// TIA Portal project "PLC_ScadaIT" (V15)

(* hardware
DEVICE "S71500/ET200MP station_1"  S7-1500 station
   slot 0: "Rail_0"  Rack  6ES7 590-1***0-0AA0
   slot 1: "PLC_CENTRAL.TAKT"  CPU 1516-3 PN/DP  6ES7 516-3AN01-0AB0  V2.5
      slot 3: "CPU display_1"  6ES7591-1BA00-0AA0
DEVICE "HMI_CENTRAL.TAKT"  TP900 Comfort
   slot 0: "HMI"  HMI  6AV2 124-0JC01-0AX0  13.0.1.0
   slot 1: "HMI_RT_1"  TP900 Comfort  6AV2 124-0JC01-0AX0  13.0.1.0
   slot 5: "HMI_CENTRAL.TAKT.IE_CP_1"  PROFINET Interface
      slot 1: "PROFINET Interface_1"  PROFINET Interface
         slot 1: "Port_1"  Port
         slot 2: "Port_2"  Port
   slot 7: "HMI_CENTRAL.TAKT.MPI/DP_CP_1"  MPI/DP Interface
*)

// ===== PLC "PLC_CENTRAL.TAKT"  CPU 1516-3 PN/DP =====

VAR_GLOBAL   // PLC tag table "Default tag table"
   "Clock_Byte" AT %MB0 : Byte;   // Byte de Clock
   "Clock_10Hz" AT %M0.0 : Bool;   // 0.1 Segundo
   "Clock_5Hz" AT %M0.1 : Bool;   // 0.2 Segundo
   "Clock_2.5Hz" AT %M0.2 : Bool;   // 0.4 Segundo
   "Clock_2Hz" AT %M0.3 : Bool;   // 0.5 Segundo
   "Clock_1.25Hz" AT %M0.4 : Bool;   // 0.8 Segundo
   "Clock_1Hz" AT %M0.5 : Bool;   // 1.0 Segundo
   "Clock_0.625Hz" AT %M0.6 : Bool;   // 1.6 Segundo
   "Clock_0.5Hz" AT %M0.7 : Bool;   // 2 Segundo
   "OFF" AT %M1.0 : Bool;   // First Scan
   "STATUS_PUT_DOCK" AT %MW603 : Word;
   "System_Byte" AT %MB1 : Byte;
   "DiagStatusUpdate" AT %M1.1 : Bool;
   "AlwaysTRUE" AT %M1.2 : Bool;
   "AlwaysFALSE" AT %M1.3 : Bool;
   "JOOJ" AT %M2.0 : Bool;
END_VAR

TYPE "Line_ReadInformation"
VERSION : 0.1
   STRUCT
      AndonExterno : Bool;   // Sinal recebido via sistema (celular)
      AndonP1 : Bool;   // Botão de andon do posto 1
      AndonP2 : Bool;   // Botão de andon do posto 2
      AndonP3 : Bool;   // Botão de andon do posto 3
      AndonP4 : Bool;   // Botão de andon do posto 4
      AndonP5 : Bool;   // Botão de andon do posto 5
      AndonP6 : Bool;   // Botão de andon do posto 6
      SensorFimDeLinha : Bool;   // Sensor RetroReflexivo do último posto
      EmergênciaP1 : Bool;   // Botão de emergência do posto 1
      EmergênciaP2 : Bool;   // Botão de emergência do posto 2
      EmergênciaP3 : Bool;   // Botão de emergência do posto 3
      EmergênciaP4 : Bool;   // Botão de emergência do posto 4
      EmergênciaP5 : Bool;   // Botão de emergência do posto 5
      EmergênciaP6 : Bool;   // Botão de emergência do posto 6
      StartRecebido : Bool;   // Confirma o recebimento do sinal de start
   END_STRUCT;
END_TYPE

TYPE "Agv.Database"
   STRUCT
      Emergencia : Bool;   // Botao de Emergecencia
      Warning : Bool;   // Area de Warning do Scanner
      Safety : Bool;   // Area de Safety do Scanner
      ConectarTakt : Bool;   // 0 - Desconectado / 1 - Conectado
      Rodando : Bool;
      Falha : Bool;
      AutomaticoManual : Byte;   // 1 - Manual / 2 - Automatico
      VelocidadeAtual : Int;   // Velocidade Atual
      Posto : Byte;   // Posto em que o AGV está
      Comando : Byte;   // Ultimo comando
      Velocidade : Byte;   // Velocidade Setada
      Processo : Byte;   // 1 - Ecu / 2 - SKD
      "Erros.Agv" : Byte;   // 0 á 256, cada numero um erro. 1 - Tudo Ok
      "Erros.Pgv" : Byte;   // 0 á 256, cada numero um erro. 1 - Tudo Ok
      "Erros.Rfid" : Byte;   // 0 á 256, cada numero um erro. 1 - Tudo Ok
      "Erros.MotorPasso" : Byte;   // 0 á 256, cada numero um erro. 1 - Tudo Ok
      "Erros.IOLink" : Byte;   // 0 á 256, cada numero um erro. 1 - Tudo Ok
      "Erros.Comunicacao" : Byte;   // 0 á 256, cada numero um erro. 1 - Tudo Ok
      Reservado : Byte;   // Reservado
      Reservado_1 : Byte;   // Reservado
      Reservado_2 : Byte;   // Reservado
      Reservado_3 : Byte;   // Reservado
      Reservado_4 : Byte;   // Reservado
      Reservado_5 : Byte;   // Reservado
      Reservado_6 : Byte;   // Reservado
      Reservado_7 : Byte;   // Reservado
      Reservado_8 : Byte;   // Reservado
   END_STRUCT;
END_TYPE

TYPE "Scada.Datebase"
   STRUCT
      Turnos : Struct
         Inicio : Array[0..2] of Time_Of_Day;
         Fim : Array[0..2] of Time_Of_Day;
      END_STRUCT;
      Paradas_Programadas : Struct
         Inicio : Array[0..5] of Time_Of_Day;
         Fim : Array[0..5] of Time_Of_Day;
      END_STRUCT;
      Dias_Da_Semana : Array[0..6] of Bool;
      ParametrosTakt : Array[0..2] of Struct
         Tempo_Takt : Int;
         ObjetivoTurno : Int;
      END_STRUCT;
      DiaDaSemana : Int;
   END_STRUCT;
   // // Dias_Da_Semana[0] : Segunda-Feira
   // // Dias_Da_Semana[1] : Terça-Feira
   // // Dias_Da_Semana[2] : Quarta-Feira
   // // Dias_Da_Semana[3] : Quinta-Feira
   // // Dias_Da_Semana[4] : Sexta-Feira
   // // Dias_Da_Semana[5] : Sabado
   // // Dias_Da_Semana[6] : Domingo
   // // ParametrosTakt[0] : Parametros do Takt do 1 turno
   // // ParametrosTakt[1] : Parametros do Takt do 2 turno
   // // ParametrosTakt[2] : Parametros do Takt do 3 turno
   // // Turnos.Inicio[0] : Incio 1 Turno
   // // Turnos.Inicio[1] : Incio 2 Turno
   // // Turnos.Inicio[2] : Incio 3 Turno
   // // Turnos.Fim[0] : Fim 1 Turno
   // // Turnos.Fim[1] : Fim 2 Turno
   // // Turnos.Fim[2] : Fim 3 Turno
   // // Paradas_Programadas.Inicio[0] : Inicio Parada Programada 1
   // // Paradas_Programadas.Inicio[1] : Inicio Parada Programada 2
   // // Paradas_Programadas.Fim[0] : Fim Parada Programada 1
   // // Paradas_Programadas.Inicio[2] : Inicio Parada Programada 3
   // // Paradas_Programadas.Inicio[3] : Inicio Parada Programada 4
   // // Paradas_Programadas.Inicio[4] : Inicio Parada Programada 5
   // // Paradas_Programadas.Inicio[5] : Inicio Parada Programada 6
   // // Paradas_Programadas.Fim[1] : Fim Parada Programada 2
   // // Paradas_Programadas.Fim[2] : Fim Parada Programada 3
   // // Paradas_Programadas.Fim[3] : Fim Parada Programada 4
   // // Paradas_Programadas.Fim[4] : Fim Parada Programada 5
   // // Paradas_Programadas.Fim[5] : Fim Parada Programada 6
END_TYPE

TYPE "AGV_READ.INFORMATION"
VERSION : 0.1
   STRUCT
      CURRENTLY_STATION : Int;
      STOP_BUTTON : Bool;
      ANDON : Bool;
      SCANNER_SAFETY : Bool;
      MOVING : Bool;
      FAULT : Bool;
      empty1 : Bool;
      empty2 : Bool;
      empty3 : Bool;
      empty4 : Bool;
      empty5 : Bool;
      empty6 : Bool;
      empty7 : Bool;
      empty8 : Bool;
      empty9 : Bool;
      empty10 : Bool;
      empty11 : Bool;
      FAULT_NUMBER : Int;
      WATCH_DOG : Int;
   END_STRUCT;
END_TYPE

TYPE "TAKT_OUTPUT.INFORMATION"
VERSION : 0.1
   STRUCT
      TAKT_ET : Int;   // Takt
      STOP_TIME : Int;   // Stop time
      ACTUAL_PRODUCTION : Int;   // Acutal production
      TARGET : Int;   // Target
      ANDON : Byte;   // Andon Button
      EMERGENCY : Byte;   // Emergency button
      "FAULT.NUMBER" : Array[1..7] of Byte;
      "BREAK.ACTUAL" : Int;
   END_STRUCT;
END_TYPE

TYPE "Central.Database"
   STRUCT
      Dados_Agv : Array[0..12] of "Agv.Database";
      Dados_Takt : Struct
         Tempo_Takt : DInt;
         Tempo_StopTime : DInt;
         Objetivo : Int;
         Atual : Int;
         TempoParada : DInt;
         Andons : Array[0..8] of Bool;
      END_STRUCT;
      Dados_Paradas : Array[0..20] of "UltimasParadas";
   END_STRUCT;
END_TYPE

TYPE "DadosDosTakts"
   STRUCT
      Linhas_Cabinas : Struct   // Linha de Cabinas
         Tempo_Takt : DInt;   // Tempo do Timer do Takt
         Tempo_StopTime : DInt;   // Tempo do Timer do Stop TIme
         Objetivo : Int;   // Objetivo de produção do dia
         Atual : Int;   // Produção atual
         LinhaParada : Bool;   // 0 - Linha está sem parada programada / 1 - Linha está em parada programada
         TempoRetornoParada : DInt;   // Tempo regressivo para o proximo turno ou re-inicio do turno
         LinhaRodando : Bool;   // 0 - Linha parada / 1 - Linha rodando
         Andons : Array[0..8] of Bool;   // Andons 0 - não acionados / 1 - Acionados
         CorDeTela : Byte;   // Cor da tela: 0 - Branco/Preto, 1 - Amarelo, 2 - Vermelho, 3 Azul, 4 - Laranja
         DirectRun : Real;   // Calculo do Direct Run
         SaldoDoTurno : Int;   // Saldo negativo do Turno
         AndonOn : Int;   // Momento em que o Andon foi acionado
         Paradas : Array[0..1] of Struct   // 2 ultimas paradas por andon
            Inicio : Time_Of_Day;   // Inicio da parada
            Fim : Time_Of_Day;   // Fim da parada
            Posto : Int;   // Posto que parau
            ValorTimer : Int;   // Valor do Timer quando parou
            ValorTimerFim : Int;   // Valor do Timer quando voltou
         END_STRUCT;
         NumMensagem : Int;   // Numero da mensagem de falha
         Emergencias : Array[0..8] of Bool;
      END_STRUCT;
      Mensagem_Cab : String;
      Linhas_SKD : Struct   // Linha de desmontagem - SKD
         Tempo_Takt : DInt;   // Tempo do Timer do Takt
         Tempo_StopTime : DInt;   // Tempo do Timer do Stop TIme
         Objetivo : Int;   // Objetivo de produção do dia
         Atual : Int;   // Produção atual
         LinhaParada : Bool;   // 0 - Linha está sem parada programada / 1 - Linha está em parada programada
         TempoRetornoParada : DInt;   // Tempo regressivo para o proximo turno ou re-inicio do turno
         LinhaRodando : Bool;   // 0 - Linha parada / 1 - Linha rodando
         Andons : Array[0..8] of Bool;   // Andons 0 - não acionados / 1 - Acionados
         CorDeTela : Byte;   // Cor da tela: 0 - Branco/Preto, 1 - Amarelo, 2 - Vermelho, 3 Azul, 4 - Laranja
         DirectRun : Real;   // Calculo do Direct Run
         SaldoDoTurno : Int;   // Saldo negativo do Turno
         AndonOn : Int;   // Momento em que o Andon foi acionado
         Paradas : Array[0..1] of Struct   // 2 ultimas paradas por andon
            Inicio : Time_Of_Day;   // Inicio da parada
            Fim : Time_Of_Day;   // Fim da parada
            Posto : Int;   // Posto que parau
            ValorTimer : Int;   // Valor do Timer quando parou
            ValorTimerFim : Int;   // Valor do Timer quando voltou
         END_STRUCT;
         NumMensagem : Int;   // Numero da mensagem de falha
         Emergencias : Array[0..8] of Bool;
      END_STRUCT;
      Mensagem_Skd : String;
      Linhas_EixoMotor : Struct   // Linha de Componentes Eixo Motor
         Tempo_Takt : DInt;   // Tempo do Timer do Takt
         Tempo_StopTime : DInt;   // Tempo do Timer do Stop TIme
         Objetivo : Int;   // Objetivo de produção do dia
         Atual : Int;   // Produção atual
         LinhaParada : Bool;   // 0 - Linha está sem parada programada / 1 - Linha está em parada programada
         TempoRetornoParada : DInt;   // Tempo regressivo para o proximo turno ou re-inicio do turno
         LinhaRodando : Bool;   // 0 - Linha parada / 1 - Linha rodando
         Andons : Array[0..8] of Bool;   // Andons 0 - não acionados / 1 - Acionados
         CorDeTela : Byte;   // Cor da tela: 0 - Branco/Preto, 1 - Amarelo, 2 - Vermelho, 3 Azul, 4 - Laranja
         DirectRun : Real;   // Calculo do Direct Run
         SaldoDoTurno : Int;   // Saldo negativo do Turno
         AndonOn : Int;   // Momento em que o Andon foi acionado
         Paradas : Array[0..1] of Struct   // 2 ultimas paradas por andon
            Inicio : Time_Of_Day;   // Inicio da parada
            Fim : Time_Of_Day;   // Fim da parada
            Posto : Int;   // Posto que parau
            ValorTimer : Int;   // Valor do Timer quando parou
            ValorTimerFim : Int;   // Valor do Timer quando voltou
         END_STRUCT;
         NumMensagem : Int;   // Numero da mensagem de falha
         Emergencias : Array[0..8] of Bool;
      END_STRUCT;
      Mensagem_Comp : String;
      Linhas_ECU : Struct   // Linha de Embalagem do motor/ ECU
         Tempo_Takt : DInt;   // Tempo do Timer do Takt
         Tempo_StopTime : DInt;   // Tempo do Timer do Stop TIme
         Objetivo : Int;   // Objetivo de produção do dia
         Atual : Int;   // Produção atual
         LinhaParada : Bool;   // 0 - Linha está sem parada programada / 1 - Linha está em parada programada
         TempoRetornoParada : DInt;   // Tempo regressivo para o proximo turno ou re-inicio do turno
         LinhaRodando : Bool;   // 0 - Linha parada / 1 - Linha rodando
         Andons : Array[0..8] of Bool;   // Andons 0 - não acionados / 1 - Acionados
         CorDeTela : Byte;   // Cor da tela: 0 - Branco/Preto, 1 - Amarelo, 2 - Vermelho, 3 Azul, 4 - Laranja
         DirectRun : Real;   // Calculo do Direct Run
         SaldoDoTurno : Int;   // Saldo negativo do Turno
         AndonOn : Int;   // Momento em que o Andon foi acionado
         Paradas : Array[0..1] of Struct   // 2 ultimas paradas por andon
            Inicio : Time_Of_Day;   // Inicio da parada
            Fim : Time_Of_Day;   // Fim da parada
            Posto : Int;   // Posto que parau
            ValorTimer : Int;   // Valor do Timer quando parou
            ValorTimerFim : Int;   // Valor do Timer quando voltou
         END_STRUCT;
         NumMensagem : Int;   // Numero da mensagem de falha
         Emergencias : Array[0..8] of Bool;
      END_STRUCT;
      Mensagem_Ecu : String;
      Docas_Estufagem : Array[0..3] of Struct
         Tempo_Takt : DInt;   // Tempo do Timer do Takt
         Tempo_StopTime : DInt;   // Tempo do Timer do Stop TIme
         Objetivo : Int;   // Tempo do Timer do Takt
         Atual : Int;   // Tempo do Timer do Stop TIme
         LinhaParada : Bool;   // Objetivo de produção do dia
         TempoRetornoParada : DInt;   // Produção atual
         LinhaRodando : Bool;   // 0 - Linha está sem parada programada / 1 - Linha está em parada programada
         Andons : Array[0..8] of Bool;   // Tempo regressivo para o proximo turno ou re-inicio do turno
         CorDeTela : Byte;   // 0 - Linha parada / 1 - Linha rodando
         DirectRun : Real;   // Andons 0 - não acionados / 1 - Acionados
         SaldoDoTurno : Int;   // Cor da tela: 0 - Branco/Preto, 1 - Amarelo, 2 - Vermelho, 3 Azul, 4 - Laranja
         AndonOn : Int;   // Calculo do Direct Run
         Paradas : Array[0..1] of Struct   // Saldo negativo do Turno
            Inicio : Time_Of_Day;   // Inicio da parada
            Fim : Time_Of_Day;   // Fim da parada
            Posto : Int;   // Posto que parau
            ValorTimer : Int;   // Valor do Timer quando parou
            ValorTimerFim : Int;   // Valor do Timer quando voltou
         END_STRUCT;
         NumMensagem : Int;   // Momento em que o Andon foi acionado
         Emergencias : Array[0..8] of Bool;
      END_STRUCT;
   END_STRUCT;
END_TYPE

TYPE "SistemaToTakt"
   STRUCT
      Inicio : Array[0..4] of Int;
      Fim : Array[0..4] of Int;
      Takt : Int;
      Objetivo : Int;
      Turno : Int;
      Refeicao : Array[0..4] of Int;
      Parada : Bool;
      Gap : Bool;
      Paradas : Array[0..4] of Struct
         Inicio : Array[0..4] of Int;
         Fim : Array[0..4] of Int;
      END_STRUCT;
   END_STRUCT;
   // // Inicio[0] : Ano
   // // Inicio[1] : Mês
   // // Inicio[2] : Dia
   // // Inicio[3] : Hora
   // // Inicio[4] : Minuto
   // // Fim[0] : Ano
   // // Fim[1] : Mês
   // // Fim[2] : Dia
   // // Fim[3] : Hora
   // // Fim[4] : Minuto
   // // Refeicao[0] : Ano
   // // Refeicao[1] : Mês
   // // Refeicao[2] : Dia
   // // Refeicao[3] : Hora
   // // Refeicao[4] : Minuto
   // // Paradas[0].Inicio[0] : Ano
   // // Paradas[0].Inicio[1] : Mês
   // // Paradas[0].Inicio[2] : Dia
   // // Paradas[0].Inicio[3] : Hora
   // // Paradas[0].Inicio[4] : Minuto
   // // Paradas[0].Fim[0] : Ano
   // // Paradas[0].Fim[1] : Mês
   // // Paradas[0].Fim[2] : Dia
   // // Paradas[0].Fim[3] : Hora
   // // Paradas[0].Fim[4] : Minuto
END_TYPE

TYPE "Scada.Maquinas"
   STRUCT
      DadosAgvs : Array[0..12] of "Agv.Database";
   END_STRUCT;
END_TYPE

TYPE "UltimasParadas"
   STRUCT
      NumeroPosto : Int;
      InicioParada : Time_Of_Day;
      FimParada : Time_Of_Day;
      DiaDaParada : Date;
   END_STRUCT;
END_TYPE

TYPE "ScadaToLine"
   STRUCT
      Inicio : DTL;
      Fim : DTL;
      RefeicaoInicio : DTL;
      RefeicaoFim : DTL;
      Paradas : Array[0..4] of Struct
         Inicio : DTL;
         Fim : DTL;
      END_STRUCT;
   END_STRUCT;
END_TYPE

DATA_BLOCK "Teste"   // DB1
{ S7_Optimized_Access := 'FALSE' }
VERSION : 0.1
   VAR
      Frente : Bool;
      Tras : Bool;
      Esquerda : Bool;
      Direita : Bool;
   END_VAR
BEGIN
END_DATA_BLOCK

// folder: 01_Comunicacao/02_DB

DATA_BLOCK "DB100_CentralAgv_Comunicacao"   // DB100
{ S7_Optimized_Access := 'TRUE' }
AUTHOR : ssbjvq
VERSION : 0.1
// stored: InstanceOfName FB100_CentralAgv_Comunicacao
"FB100_CentralAgv_Comunicacao"
BEGIN
END_DATA_BLOCK

DATA_BLOCK "DB101_ComunicacaoEscravos"   // DB101
{ S7_Optimized_Access := 'TRUE' }
VERSION : 0.1
// stored: InstanceOfName FB101_ComunicacaoEscravos
"FB101_ComunicacaoEscravos"
BEGIN
END_DATA_BLOCK

DATA_BLOCK "DB103_DadosCabLine"   // DB103
{ S7_Optimized_Access := 'FALSE' }
VERSION : 0.1
   VAR
      "CAB.LINEFEEDING" : "TAKT_OUTPUT.INFORMATION";
      "CAB.MAINLINE" : "TAKT_OUTPUT.INFORMATION";
      "CAB.CONTAINERSTUFFING" : "TAKT_OUTPUT.INFORMATION";
   END_VAR
BEGIN
END_DATA_BLOCK

DATA_BLOCK "DB104_DadosSkdLine"   // DB104
TITLE = DB104_DadosSkdLine
{ S7_Optimized_Access := 'FALSE' }
VERSION : 0.1
   VAR
      "SKD.LINEFEEDING" : "TAKT_OUTPUT.INFORMATION";
      "SKD.MAINLINE" : "TAKT_OUTPUT.INFORMATION";
      "SKD.CONTAINERSTUFFING" : "TAKT_OUTPUT.INFORMATION";
   END_VAR
BEGIN
END_DATA_BLOCK

DATA_BLOCK "DB105_DadosCompLine"   // DB105
TITLE = DB105_DadosCompLine
{ S7_Optimized_Access := 'FALSE' }
VERSION : 0.1
   VAR
      "SKID.LINEFEEDING" : "TAKT_OUTPUT.INFORMATION";
      "SKID.MAINLINE" : "TAKT_OUTPUT.INFORMATION";
      "SKID.CONTAINERSTUFFING" : "TAKT_OUTPUT.INFORMATION";
   END_VAR
BEGIN
END_DATA_BLOCK

DATA_BLOCK "DB106_DadosEcuLine"   // DB106
{ S7_Optimized_Access := 'FALSE' }
VERSION : 0.1
   VAR
      "AGV.LINEFEEDING" : "TAKT_OUTPUT.INFORMATION";
      "AGV.MAINLINE" : "TAKT_OUTPUT.INFORMATION";
      "AGV.CONTAINERSTUFFING" : "TAKT_OUTPUT.INFORMATION";
   END_VAR
BEGIN
END_DATA_BLOCK

DATA_BLOCK "DB107_EnviaDados_DB"   // DB107
{ S7_Optimized_Access := 'TRUE' }
VERSION : 0.1
// stored: InstanceOfName FB107_EnviaDados
"FB107_EnviaDados"
BEGIN
END_DATA_BLOCK

// folder: 02_Takt/02_DB

DATA_BLOCK "DB201_FiltragemDados"   // DB201
{ S7_Optimized_Access := 'TRUE' }
VERSION : 0.1
// stored: InstanceOfName FB201_FiltragemDados
"FB201_FiltragemDados"
BEGIN
END_DATA_BLOCK

DATA_BLOCK "DB206_CheckEmTurno"   // DB206
{ S7_Optimized_Access := 'TRUE' }
VERSION : 0.1
// stored: InstanceOfName FB206_CheckEmTurno
"FB206_CheckEmTurno"
BEGIN
END_DATA_BLOCK

DATA_BLOCK "DB207_ConcatAgvData"   // DB207
{ S7_Optimized_Access := 'TRUE' }
VERSION : 0.1
// stored: InstanceOfName FB207_ConcatAgvData
"FB207_ConcatAgvData"
BEGIN
END_DATA_BLOCK

DATA_BLOCK "DB208_ConcatLinhasData"   // DB208
{ S7_Optimized_Access := 'TRUE' }
VERSION : 0.1
// stored: InstanceOfName FB208_ConcatLinhasData
"FB208_ConcatLinhasData"
BEGIN
END_DATA_BLOCK

DATA_BLOCK "DB209_FormatadorDados"   // DB209
{ S7_Optimized_Access := 'TRUE' }
VERSION : 0.1
// stored: InstanceOfName FB209_FormatadorDados
"FB209_FormatadorDados"
BEGIN
END_DATA_BLOCK

DATA_BLOCK "DB210_SistemaToPlc"   // DB210
TITLE = DB210_SistemaToPlc
{ S7_Optimized_Access := 'FALSE' }
VERSION : 0.1
// DB210_SistemaToPlc
   VAR
      "Powertrain-Ecu" : "SistemaToTakt";
      Componentes : "SistemaToTakt";
      Skd : "SistemaToTakt";
      "Cabinas-Ecu" : "SistemaToTakt";
      Doca1 : "SistemaToTakt";
      Doca2 : "SistemaToTakt";
      Doca3 : "SistemaToTakt";
      Doca4 : "SistemaToTakt";
   END_VAR
BEGIN
END_DATA_BLOCK

DATA_BLOCK "DB211_DadosScada"   // DB211
TITLE = DB211_DadosScada
{ S7_Optimized_Access := 'FALSE' }
VERSION : 0.1
   VAR
      Cabinas : Struct
         "Timer" : Int;
         StopTime : Int;
         Objetivo : Byte;
         Atual : Byte;
         TempoRetornoParada : Int;
         Andon : Byte;
         Emergencia : Byte;
         CorDeTela : Byte;
         NumMensagem : Byte;
      END_STRUCT;
      Skd : Struct
         "Timer" : Int;
         StopTime : Int;
         Objetivo : Byte;
         Atual : Byte;
         TempoRetornoParada : Int;
         Andon : Byte;
         Emergencia : Byte;
         CorDeTela : Byte;
         NumMensagem : Byte;
      END_STRUCT;
      Comp : Struct
         "Timer" : Int;
         StopTime : Int;
         Objetivo : Byte;
         Atual : Byte;
         TempoRetornoParada : Int;
         Andon : Byte;
         Emergencia : Byte;
         CorDeTela : Byte;
         NumMensagem : Byte;
      END_STRUCT;
      Ecu : Struct
         "Timer" : Int;
         StopTime : Int;
         Objetivo : Byte;
         Atual : Byte;
         TempoRetornoParada : Int;
         Andon : Byte;
         Emergencia : Byte;
         CorDeTela : Byte;
         NumMensagem : Byte;
      END_STRUCT;
      Docas : Array[0..3] of Struct
         "Timer" : Int;
         StopTime : Int;
         Objetivo : Byte;
         Atual : Byte;
         TempoRetornoParada : Int;
         Andon : Byte;
         Emergencia : Byte;
         CorDeTela : Byte;
         NumMensagem : Byte;
      END_STRUCT;
      AGV : Array[0..9] of Struct
         Sinais : Byte;
         Posto : Byte;
         Comando : Byte;
         Velocidade : Byte;
         Processo : Byte;
         VelAtual : Byte;
         "Erros.Agv" : Byte;
         "Erros.Pgv" : Byte;
         "Erros.MotorPasso" : Byte;
      END_STRUCT;
      "Array" : Array[0..17] of String;
      Array_Byte : Array[0..30] of Byte;
   END_VAR
BEGIN
   Array_Byte[0] := 1;
   Array_Byte[1] := 2;
   Array_Byte[2] := 10;
END_DATA_BLOCK

DATA_BLOCK "DB212_FomatadorSistemaToPlc"   // DB212
{ S7_Optimized_Access := 'TRUE' }
VERSION : 0.1
// stored: InstanceOfName FB212_FomatadorSistemaToPlc
"FB212_FomatadorSistemaToPlc"
BEGIN
END_DATA_BLOCK

DATA_BLOCK "DB214_ScadaToLines"   // DB214
TITLE = DB214_ScadaToLines
{ S7_Optimized_Access := 'FALSE' }
VERSION : 0.1
   VAR
      Cabinas : Array[0..2] of "ScadaToLine";
      Skd : Array[0..2] of "ScadaToLine";
      Componentes : Array[0..2] of "ScadaToLine";
      "Powertrain-Ecu" : Array[0..2] of "ScadaToLine";
      Doca1 : Array[0..2] of "ScadaToLine";
      Doca2 : Array[0..2] of "ScadaToLine";
      Doca3 : Array[0..2] of "ScadaToLine";
      Doca4 : Array[0..2] of "ScadaToLine";
   END_VAR
BEGIN
   // Cabinas[0] : 1º Turno
   // Cabinas[1] : 2º Turno
   // Cabinas[2] : 3º Turno
   // Skd[0] : 1º Turno
   // Skd[1] : 2º Turno
   // Skd[2] : 3º Turno
   // Componentes[0] : 1º Turno
   // Componentes[1] : 2º Turno
   // Componentes[2] : 3º Turno
   // "Powertrain-Ecu"[0] : 1º Turno
   // "Powertrain-Ecu"[1] : 2º Turno
   // "Powertrain-Ecu"[2] : 3º Turno
   // Doca1[0] : 1º Turno
   // Doca1[1] : 2º Turno
   // Doca1[2] : 3º Turno
   // Doca2[0] : 1º Turno
   // Doca2[1] : 2º Turno
   // Doca2[2] : 3º Turno
   // Doca3[0] : 1º Turno
   // Doca3[1] : 2º Turno
   // Doca3[2] : 3º Turno
   // Doca4[0] : 1º Turno
   // Doca4[1] : 2º Turno
   // Doca4[2] : 3º Turno
END_DATA_BLOCK

DATA_BLOCK "DB215_SistemaToPlc_2Turno"   // DB215
TITLE = DB215_SistemaToPlc_2Turno
{ S7_Optimized_Access := 'FALSE' }
VERSION : 0.1
   VAR
      "Powertrain-Ecu" : "SistemaToTakt";
      Componentes : "SistemaToTakt";
      Skd : "SistemaToTakt";
      "Cabinas-Ecu" : "SistemaToTakt";
      Doca1 : "SistemaToTakt";
      Doca2 : "SistemaToTakt";
      Doca3 : "SistemaToTakt";
      Doca4 : "SistemaToTakt";
   END_VAR
BEGIN
END_DATA_BLOCK

DATA_BLOCK "DB216_SistemaToPlc_3Turno"   // DB216
TITLE = DB216_SistemaToPlc_3Turno
{ S7_Optimized_Access := 'FALSE' }
VERSION : 0.1
   VAR
      "Powertrain-Ecu" : "SistemaToTakt";
      Componentes : "SistemaToTakt";
      Skd : "SistemaToTakt";
      "Cabinas-Ecu" : "SistemaToTakt";
      Doca1 : "SistemaToTakt";
      Doca2 : "SistemaToTakt";
      Doca3 : "SistemaToTakt";
      Doca4 : "SistemaToTakt";
   END_VAR
BEGIN
END_DATA_BLOCK

DATA_BLOCK "DB1000_DadosDosTakts"   // DB1000
TITLE = DB1000_DadosDosTakts
{ S7_Optimized_Access := 'FALSE' }
AUTHOR : ssbjvq
VERSION : 0.1
// Está DB é responsavel por centralizar os dados dos Takts para que o sistema faça a leitura
   VAR
      Dados : "DadosDosTakts";   // Dados referente a todos os takts do KD
   END_VAR
BEGIN
END_DATA_BLOCK

// folder: 03_Ihm/02_DB

DATA_BLOCK "DB300_IhmDados"   // DB300
{ S7_Optimized_Access := 'FALSE' }
VERSION : 0.1
   VAR
      Dados_Cabinas : Struct
         Tempo_Takt : DInt;
         Tempo_StopTime : DInt;
         Objetivo : Int;
         Atual : Int;
         LinhaParada : Bool;
         TempoRetornoParada : DInt;
         LinhaRodando : Bool;
         Andons : Array[0..8] of Bool;
         CorDeTela : Byte;
         DirectRun : Real;
         SaldoDoTurno : Int;
         AndonOn : Int;
         Paradas : Array[0..1] of Struct
            Inicio : Time_Of_Day;
            Fim : Time_Of_Day;
            Posto : Int;
            ValorTimer : Int;
            ValorTimerFim : Int;
         END_STRUCT;
         NumMensagem : Int;
         Emergencias : Array[0..8] of Bool;
      END_STRUCT;
      Mensagem_Cab : String;
      Dados_SKD : Struct
         Tempo_Takt : DInt;
         Tempo_StopTime : DInt;
         Objetivo : Int;
         Atual : Int;
         LinhaParada : Bool;
         TempoRetornoParada : DInt;
         LinhaRodando : Bool;
         Andons : Array[0..8] of Bool;
         CorDeTela : Byte;
         DirectRun : Real;
         SaldoDoTurno : Int;
         AndonOn : Int;
         Paradas : Array[0..1] of Struct
            Inicio : Time_Of_Day;
            Fim : Time_Of_Day;
            Posto : Int;
            ValorTimer : Int;
            ValorTimerFim : Int;
         END_STRUCT;
         NumMensagem : Int;
         Emergencias : Array[0..8] of Bool;
      END_STRUCT;
      Mensagem_SKD : String;
      Dados_Componentes : Struct
         Tempo_Takt : DInt;
         Tempo_StopTime : DInt;
         Objetivo : Int;
         Atual : Int;
         LinhaParada : Bool;
         TempoRetornoParada : DInt;
         LinhaRodando : Bool;
         Andons : Array[0..8] of Bool;
         CorDeTela : Byte;
         DirectRun : Real;
         SaldoDoTurno : Int;
         AndonOn : Int;
         Paradas : Array[0..1] of Struct
            Inicio : Time_Of_Day;
            Fim : Time_Of_Day;
            Posto : Int;
            ValorTimer : Int;
            ValorTimerFim : Int;
         END_STRUCT;
         NumMensagem : Int;
         Emergencias : Array[0..8] of Bool;
      END_STRUCT;
      Mensagem_Componentes : String;
      Dados_ECU : Struct
         Tempo_Takt : DInt;
         Tempo_StopTime : DInt;
         Objetivo : Int;
         Atual : Int;
         LinhaParada : Bool;
         TempoRetornoParada : DInt;
         LinhaRodando : Bool;
         Andons : Array[0..8] of Bool;
         CorDeTela : Byte;
         DirectRun : Real;
         SaldoDoTurno : Int;
         AndonOn : Int;
         Paradas : Array[0..1] of Struct
            Inicio : Time_Of_Day;
            Fim : Time_Of_Day;
            Posto : Int;
            ValorTimer : Int;
            ValorTimerFim : Int;
         END_STRUCT;
         NumMensagem : Int;
         Emergencias : Array[0..8] of Bool;
      END_STRUCT;
      Mensagem_ECU : String;
   END_VAR
BEGIN
END_DATA_BLOCK

DATA_BLOCK "DB301_CentralToScada"   // DB301
TITLE = DB301_CentralToScada
{ S7_Optimized_Access := 'FALSE' }
VERSION : 0.1
// DB301_CentralToScada
   VAR
      Data : "Central.Database";
   END_VAR
BEGIN
END_DATA_BLOCK

DATA_BLOCK "DB302_InputDados"   // DB302
TITLE = DB302_InputDados
{ S7_Optimized_Access := 'FALSE' }
VERSION : 0.1
   VAR
      Ecu : Struct
         Turnos : Struct
            "1_Turno" : Struct
               Inicio : Date_And_Time;
               Fim : Date_And_Time;
               TempoTakt : Int;
               Rodadas : Int;
            END_STRUCT;
            "2_Turno" : Struct
               Inicio : Date_And_Time;
               Fim : Date_And_Time;
               TempoTakt : Int;
               Rodadas : Int;
            END_STRUCT;
            "3_Turno" : Struct
               Inicio : Date_And_Time;
               Fim : Date_And_Time;
               TempoTakt : Int;
               Rodadas : Int;
            END_STRUCT;
         END_STRUCT;
         Paradas_Programadas_1Turno : Struct
            Parada_1 : Struct
               Inicio : Time_Of_Day;
               Fim : Time_Of_Day;
            END_STRUCT;
            Parada_2 : Struct
               Inicio : Time_Of_Day;
               Fim : Time_Of_Day;
            END_STRUCT;
            Parada_3 : Struct
               Inicio : Time_Of_Day;
               Fim : Time_Of_Day;
            END_STRUCT;
            Parada_4 : Struct
               Inicio : Time_Of_Day;
               Fim : Time_Of_Day;
            END_STRUCT;
            Parada_5 : Struct
               Inicio : Time_Of_Day;
               Fim : Time_Of_Day;
            END_STRUCT;
         END_STRUCT;
         Paradas_Programadas_2Turno : Struct
            Parada_1 : Struct
               Inicio : Time_Of_Day;
               Fim : Time_Of_Day;
            END_STRUCT;
            Parada_2 : Struct
               Inicio : Time_Of_Day;
               Fim : Time_Of_Day;
            END_STRUCT;
            Parada_3 : Struct
               Inicio : Time_Of_Day;
               Fim : Time_Of_Day;
            END_STRUCT;
            Parada_4 : Struct
               Inicio : Time_Of_Day;
               Fim : Time_Of_Day;
            END_STRUCT;
            Parada_5 : Struct
               Inicio : Time_Of_Day;
               Fim : Time_Of_Day;
            END_STRUCT;
         END_STRUCT;
         Paradas_Programadas_3Turno : Struct
            Parada_1 : Struct
               Inicio : Time_Of_Day;
               Fim : Time_Of_Day;
            END_STRUCT;
            Parada_2 : Struct
               Inicio : Time_Of_Day;
               Fim : Time_Of_Day;
            END_STRUCT;
            Parada_3 : Struct
               Inicio : Time_Of_Day;
               Fim : Time_Of_Day;
            END_STRUCT;
            Parada_4 : Struct
               Inicio : Time_Of_Day;
               Fim : Time_Of_Day;
            END_STRUCT;
            Parada_5 : Struct
               Inicio : Time_Of_Day;
               Fim : Time_Of_Day;
            END_STRUCT;
         END_STRUCT;
         SistemaOn : Bool := FALSE;   // 1 - Habilidado o Input de dados pelo sistema / 0 - Input de dados pela IHM
         AtualizarDados : Bool;
      END_STRUCT;
      Cabinas : Struct
         Turnos : Struct
            "1_Turno" : Struct
               Inicio : Date_And_Time;
               Fim : Date_And_Time;
               TempoTakt : Int;
               Rodadas : Int;
            END_STRUCT;
            "2_Turno" : Struct
               Inicio : Date_And_Time;
               Fim : Date_And_Time;
               TempoTakt : Int;
               Rodadas : Int;
            END_STRUCT;
            "3_Turno" : Struct
               Inicio : Date_And_Time;
               Fim : Date_And_Time;
               TempoTakt : Int;
               Rodadas : Int;
            END_STRUCT;
         END_STRUCT;
         Paradas_Programadas_1Turno : Struct
            Parada_1 : Struct
               Inicio : Time;
               Fim : Time;
            END_STRUCT;
            Parada_2 : Struct
               Inicio : Time;
               Fim : Time;
            END_STRUCT;
            Parada_3 : Struct
               Inicio : Time;
               Fim : Time;
            END_STRUCT;
            Parada_4 : Struct
               Inicio : Time;
               Fim : Time;
            END_STRUCT;
            Parada_5 : Struct
               Inicio : Time;
               Fim : Time;
            END_STRUCT;
         END_STRUCT;
         Paradas_Programadas_2Turno : Struct
            Parada_1 : Struct
               Inicio : Time;
               Fim : Time;
            END_STRUCT;
            Parada_2 : Struct
               Inicio : Time;
               Fim : Time;
            END_STRUCT;
            Parada_3 : Struct
               Inicio : Time;
               Fim : Time;
            END_STRUCT;
            Parada_4 : Struct
               Inicio : Time;
               Fim : Time;
            END_STRUCT;
            Parada_5 : Struct
               Inicio : Time;
               Fim : Time;
            END_STRUCT;
         END_STRUCT;
         Paradas_Programadas_3Turno : Struct
            Parada_1 : Struct
               Inicio : Time;
               Fim : Time;
            END_STRUCT;
            Parada_2 : Struct
               Inicio : Time;
               Fim : Time;
            END_STRUCT;
            Parada_3 : Struct
               Inicio : Time;
               Fim : Time;
            END_STRUCT;
            Parada_4 : Struct
               Inicio : Time;
               Fim : Time;
            END_STRUCT;
            Parada_5 : Struct
               Inicio : Time;
               Fim : Time;
            END_STRUCT;
         END_STRUCT;
         SistemaOn : Bool := FALSE;   // 1 - Habilidado o Input de dados pelo sistema / 0 - Input de dados pela IHM
      END_STRUCT;
      SKD : Struct
         Turnos : Struct
            "1_Turno" : Struct
               Inicio : Date_And_Time;
               Fim : Date_And_Time;
               TempoTakt : Int;
               Rodadas : Int;
            END_STRUCT;
            "2_Turno" : Struct
               Inicio : Date_And_Time;
               Fim : Date_And_Time;
               TempoTakt : Int;
               Rodadas : Int;
            END_STRUCT;
            "3_Turno" : Struct
               Inicio : Date_And_Time;
               Fim : Date_And_Time;
               TempoTakt : Int;
               Rodadas : Int;
            END_STRUCT;
         END_STRUCT;
         Paradas_Programadas_1Turno : Struct
            Parada_1 : Struct
               Inicio : Time;
               Fim : Time;
            END_STRUCT;
            Parada_2 : Struct
               Inicio : Time;
               Fim : Time;
            END_STRUCT;
            Parada_3 : Struct
               Inicio : Time;
               Fim : Time;
            END_STRUCT;
            Parada_4 : Struct
               Inicio : Time;
               Fim : Time;
            END_STRUCT;
            Parada_5 : Struct
               Inicio : Time;
               Fim : Time;
            END_STRUCT;
         END_STRUCT;
         Paradas_Programadas_2Turno : Struct
            Parada_1 : Struct
               Inicio : Time;
               Fim : Time;
            END_STRUCT;
            Parada_2 : Struct
               Inicio : Time;
               Fim : Time;
            END_STRUCT;
            Parada_3 : Struct
               Inicio : Time;
               Fim : Time;
            END_STRUCT;
            Parada_4 : Struct
               Inicio : Time;
               Fim : Time;
            END_STRUCT;
            Parada_5 : Struct
               Inicio : Time;
               Fim : Time;
            END_STRUCT;
         END_STRUCT;
         Paradas_Programadas_3Turno : Struct
            Parada_1 : Struct
               Inicio : Time;
               Fim : Time;
            END_STRUCT;
            Parada_2 : Struct
               Inicio : Time;
               Fim : Time;
            END_STRUCT;
            Parada_3 : Struct
               Inicio : Time;
               Fim : Time;
            END_STRUCT;
            Parada_4 : Struct
               Inicio : Time;
               Fim : Time;
            END_STRUCT;
            Parada_5 : Struct
               Inicio : Time;
               Fim : Time;
            END_STRUCT;
         END_STRUCT;
         SistemaOn : Bool := FALSE;   // 1 - Habilidado o Input de dados pelo sistema / 0 - Input de dados pela IHM
      END_STRUCT;
      Componentes : Struct
         Turnos : Struct
            "1_Turno" : Struct
               Inicio : Date_And_Time;
               Fim : Date_And_Time;
               TempoTakt : Int;
               Rodadas : Int;
            END_STRUCT;
            "2_Turno" : Struct
               Inicio : Date_And_Time;
               Fim : Date_And_Time;
               TempoTakt : Int;
               Rodadas : Int;
            END_STRUCT;
            "3_Turno" : Struct
               Inicio : Date_And_Time;
               Fim : Date_And_Time;
               TempoTakt : Int;
               Rodadas : Int;
            END_STRUCT;
         END_STRUCT;
         Paradas_Programadas_1Turno : Struct
            Parada_1 : Struct
               Inicio : Time;
               Fim : Time;
            END_STRUCT;
            Parada_2 : Struct
               Inicio : Time;
               Fim : Time;
            END_STRUCT;
            Parada_3 : Struct
               Inicio : Time;
               Fim : Time;
            END_STRUCT;
            Parada_4 : Struct
               Inicio : Time;
               Fim : Time;
            END_STRUCT;
            Parada_5 : Struct
               Inicio : Time;
               Fim : Time;
            END_STRUCT;
         END_STRUCT;
         Paradas_Programadas_2Turno : Struct
            Parada_1 : Struct
               Inicio : Time;
               Fim : Time;
            END_STRUCT;
            Parada_2 : Struct
               Inicio : Time;
               Fim : Time;
            END_STRUCT;
            Parada_3 : Struct
               Inicio : Time;
               Fim : Time;
            END_STRUCT;
            Parada_4 : Struct
               Inicio : Time;
               Fim : Time;
            END_STRUCT;
            Parada_5 : Struct
               Inicio : Time;
               Fim : Time;
            END_STRUCT;
         END_STRUCT;
         Paradas_Programadas_3Turno : Struct
            Parada_1 : Struct
               Inicio : Time;
               Fim : Time;
            END_STRUCT;
            Parada_2 : Struct
               Inicio : Time;
               Fim : Time;
            END_STRUCT;
            Parada_3 : Struct
               Inicio : Time;
               Fim : Time;
            END_STRUCT;
            Parada_4 : Struct
               Inicio : Time;
               Fim : Time;
            END_STRUCT;
            Parada_5 : Struct
               Inicio : Time;
               Fim : Time;
            END_STRUCT;
         END_STRUCT;
         SistemaOn : Bool := FALSE;   // 1 - Habilidado o Input de dados pelo sistema / 0 - Input de dados pela IHM
      END_STRUCT;
   END_VAR
BEGIN
END_DATA_BLOCK

DATA_BLOCK "DB303_ScadaToCentral"   // DB303
TITLE = DB300_MestreToCentral
{ S7_Optimized_Access := 'FALSE' }
VERSION : 0.1
// DB300_MestreToCentral
   VAR
      Data : "Scada.Datebase";
   END_VAR
BEGIN
   Data.Paradas_Programadas.Inicio[0] := TOD#11:15:00;
   Data.Paradas_Programadas.Fim[0] := TOD#12:15:00;
   Data.Turnos.Inicio[0] := TOD#07:15:00;
   Data.Turnos.Fim[0] := TOD#16:00:00;
   Data.Dias_Da_Semana[0] := TRUE;
   Data.Dias_Da_Semana[1] := TRUE;
   Data.Dias_Da_Semana[2] := TRUE;
   Data.Dias_Da_Semana[3] := TRUE;
   Data.Dias_Da_Semana[4] := TRUE;
   Data.ParametrosTakt[0].Tempo_Takt := 720;
   Data.ParametrosTakt[0].ObjetivoTurno := 48;
   Data.ParametrosTakt[1].Tempo_Takt := 720;
   Data.ParametrosTakt[1].ObjetivoTurno := 48;
   Data.ParametrosTakt[2].Tempo_Takt := 720;
   Data.ParametrosTakt[2].ObjetivoTurno := 48;
END_DATA_BLOCK

// folder: System blocks/Program resources

DATA_BLOCK "PLC_CENTRAL.TAKT_Send_DB_2"   // DB5
{ S7_Optimized_Access := 'TRUE' }
AUTHOR : SIMATIC
FAMILY : MC7Plus
NAME : TC_IP_v4
VERSION : 1.0
// stored: InstanceOfName TCON_IP_v4
"TCON_IP_v4"
BEGIN
   ID := 1;
   InterfaceId := 72;
   RemotePort := 11000;
   ActiveEstablished := true;
   RemoteAddress.ADDR[1] := 10;
   RemoteAddress.ADDR[2] := 8;
   RemoteAddress.ADDR[3] := 77;
   RemoteAddress.ADDR[4] := 65;
   ConnectionType := 11;
END_DATA_BLOCK

DATA_BLOCK "PLC_CENTRAL.TAKT_Send_DB_1"   // DB9
{ S7_Optimized_Access := 'TRUE' }
VERSION : 0.1
// stored: InstanceOfName TCON_Configured
"TCON_Configured"
BEGIN
   ID := 262;
   ConnectionType := 254;
END_DATA_BLOCK

// folder: (top level)

ORGANIZATION_BLOCK "Main"   // OB1, LAD, ProgramCycle
TITLE = "Main Program Sweep (Cycle)"
{ S7_Optimized_Access := 'TRUE' }
VERSION : 0.1
   VAR_INPUT
      Initial_Call : Bool;   // Initial call of this OB
      Remanence : Bool;   // =True, if remanent data are available
   END_VAR
   VAR_TEMP
      retval : Int;
   END_VAR
BEGIN

REGION Network 1: Bloco de comunicação com os escravos
   // Este bloco realiza a leitura dos dados dos escravos da rede
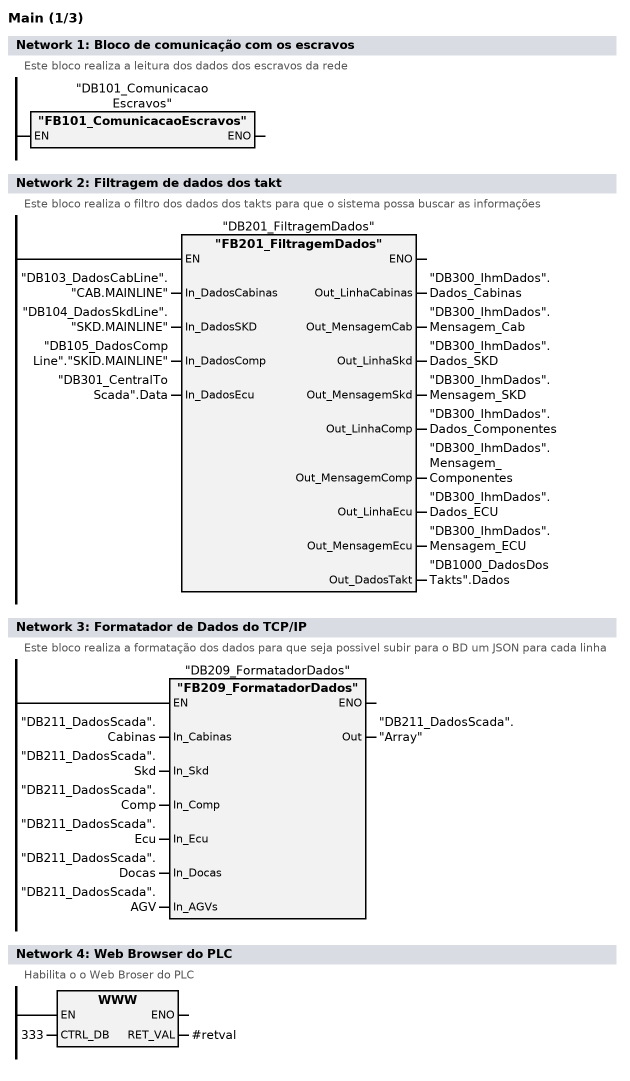
   RUNG wire#powerrail
      "DB101_ComunicacaoEscravos"()
   END_RUNG
   // the same network as SCL:
   "DB101_ComunicacaoEscravos"();   // "FB101_ComunicacaoEscravos"
END_REGION

REGION Network 2: Filtragem de dados dos takt
   // Este bloco realiza o filtro dos dados dos takts para que o sistema possa buscar as informações
   RUNG wire#powerrail
      "DB201_FiltragemDados"(In_DadosCabinas := "DB103_DadosCabLine"."CAB.MAINLINE", In_DadosSKD := "DB104_DadosSkdLine"."SKD.MAINLINE", In_DadosComp := "DB105_DadosCompLine"."SKID.MAINLINE", In_DadosEcu := "DB301_CentralToScada".Data, Out_LinhaCabinas => "DB300_IhmDados".Dados_Cabinas, Out_MensagemCab => "DB300_IhmDados".Mensagem_Cab, Out_LinhaSkd => "DB300_IhmDados".Dados_SKD, Out_MensagemSkd => "DB300_IhmDados".Mensagem_SKD, Out_LinhaComp => "DB300_IhmDados".Dados_Componentes, Out_MensagemComp => "DB300_IhmDados".Mensagem_Componentes, Out_LinhaEcu => "DB300_IhmDados".Dados_ECU, Out_MensagemEcu => "DB300_IhmDados".Mensagem_ECU, Out_DadosTakt => "DB1000_DadosDosTakts".Dados)
   END_RUNG
   // the same network as SCL:
   "DB201_FiltragemDados"(In_DadosCabinas := "DB103_DadosCabLine"."CAB.MAINLINE",   // "FB201_FiltragemDados"
                          In_DadosSKD := "DB104_DadosSkdLine"."SKD.MAINLINE",
                          In_DadosComp := "DB105_DadosCompLine"."SKID.MAINLINE",
                          In_DadosEcu := "DB301_CentralToScada".Data,
                          Out_LinhaCabinas => "DB300_IhmDados".Dados_Cabinas,
                          Out_MensagemCab => "DB300_IhmDados".Mensagem_Cab,
                          Out_LinhaSkd => "DB300_IhmDados".Dados_SKD,
                          Out_MensagemSkd => "DB300_IhmDados".Mensagem_SKD,
                          Out_LinhaComp => "DB300_IhmDados".Dados_Componentes,
                          Out_MensagemComp => "DB300_IhmDados".Mensagem_Componentes,
                          Out_LinhaEcu => "DB300_IhmDados".Dados_ECU,
                          Out_MensagemEcu => "DB300_IhmDados".Mensagem_ECU,
                          Out_DadosTakt => "DB1000_DadosDosTakts".Dados);
END_REGION

REGION Network 3: Formatador de Dados do TCP/IP
   // Este bloco realiza a formatação dos dados para que seja possivel subir para o BD um JSON para cada linha
   RUNG wire#powerrail
      "DB209_FormatadorDados"(In_Cabinas := "DB211_DadosScada".Cabinas, In_Skd := "DB211_DadosScada".Skd, In_Comp := "DB211_DadosScada".Comp, In_Ecu := "DB211_DadosScada".Ecu, In_Docas := "DB211_DadosScada".Docas, In_AGVs := "DB211_DadosScada".AGV, Out => "DB211_DadosScada"."Array")
   END_RUNG
   // the same network as SCL:
   "DB209_FormatadorDados"(In_Cabinas := "DB211_DadosScada".Cabinas,   // "FB209_FormatadorDados"
                           In_Skd := "DB211_DadosScada".Skd,
                           In_Comp := "DB211_DadosScada".Comp,
                           In_Ecu := "DB211_DadosScada".Ecu,
                           In_Docas := "DB211_DadosScada".Docas,
                           In_AGVs := "DB211_DadosScada".AGV,
                           Out => "DB211_DadosScada"."Array");
END_REGION

REGION Network 4: Web Browser do PLC
   // Habilita o o Web Broser do PLC
   #retval := WWW(CTRL_DB := 333);
END_REGION

REGION Network 5: Comunicação via TCP/IP
   // Envia as informações via TCP/IP para o Servidor C#
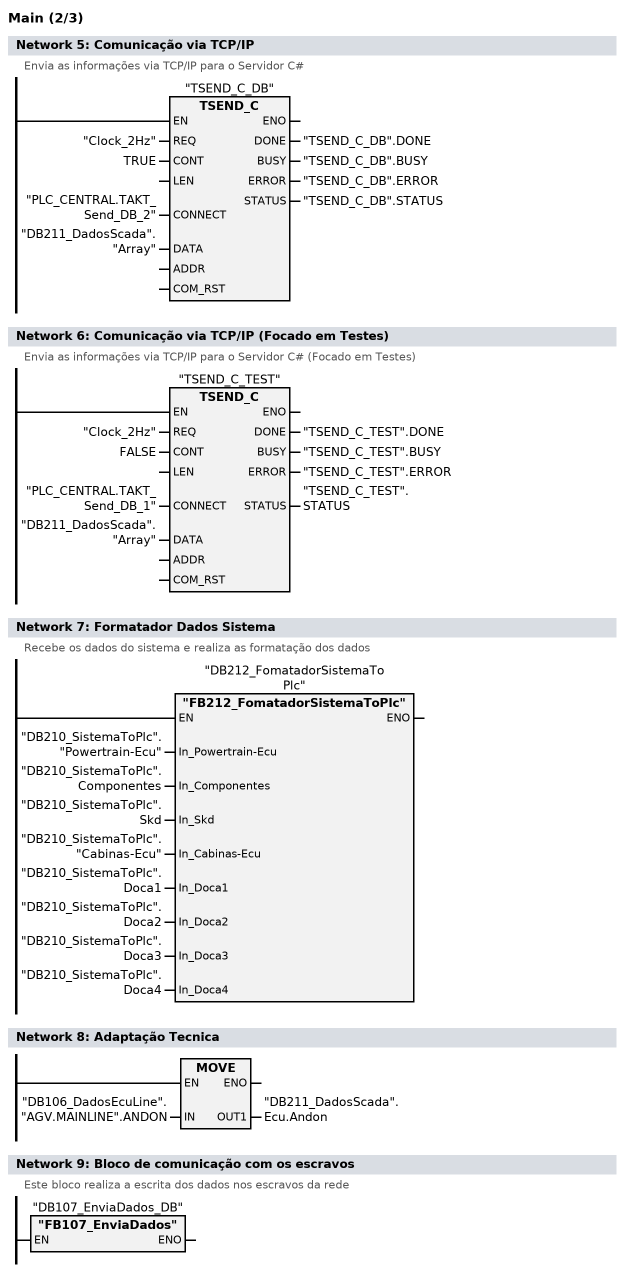
   "TSEND_C_DB"(REQ := "Clock_2Hz",   // TSEND_C
                CONT := TRUE,
                CONNECT := "PLC_CENTRAL.TAKT_Send_DB_2",
                DATA := "DB211_DadosScada"."Array",
                DONE => "TSEND_C_DB".DONE,
                BUSY => "TSEND_C_DB".BUSY,
                ERROR => "TSEND_C_DB".ERROR,
                STATUS => "TSEND_C_DB".STATUS);
END_REGION

REGION Network 6: Comunicação via TCP/IP (Focado em Testes)
   // Envia as informações via TCP/IP para o Servidor C# (Focado em Testes)
   "TSEND_C_TEST"(REQ := "Clock_2Hz",   // TSEND_C
                  CONT := FALSE,
                  CONNECT := "PLC_CENTRAL.TAKT_Send_DB_1",
                  DATA := "DB211_DadosScada"."Array",
                  DONE => "TSEND_C_TEST".DONE,
                  BUSY => "TSEND_C_TEST".BUSY,
                  ERROR => "TSEND_C_TEST".ERROR,
                  STATUS => "TSEND_C_TEST".STATUS);
END_REGION

REGION Network 7: Formatador Dados Sistema
   // Recebe os dados do sistema e realiza as formatação dos dados
   RUNG wire#powerrail
      "DB212_FomatadorSistemaToPlc"("In_Powertrain-Ecu" := "DB210_SistemaToPlc"."Powertrain-Ecu", In_Componentes := "DB210_SistemaToPlc".Componentes, In_Skd := "DB210_SistemaToPlc".Skd, "In_Cabinas-Ecu" := "DB210_SistemaToPlc"."Cabinas-Ecu", In_Doca1 := "DB210_SistemaToPlc".Doca1, In_Doca2 := "DB210_SistemaToPlc".Doca2, In_Doca3 := "DB210_SistemaToPlc".Doca3, In_Doca4 := "DB210_SistemaToPlc".Doca4)
   END_RUNG
   // the same network as SCL:
   "DB212_FomatadorSistemaToPlc"("In_Powertrain-Ecu" := "DB210_SistemaToPlc"."Powertrain-Ecu",   // "FB212_FomatadorSistemaToPlc"
                           In_Componentes := "DB210_SistemaToPlc".Componentes,
                           In_Skd := "DB210_SistemaToPlc".Skd,
                           "In_Cabinas-Ecu" := "DB210_SistemaToPlc"."Cabinas-Ecu",
                           In_Doca1 := "DB210_SistemaToPlc".Doca1,
                           In_Doca2 := "DB210_SistemaToPlc".Doca2,
                           In_Doca3 := "DB210_SistemaToPlc".Doca3,
                           In_Doca4 := "DB210_SistemaToPlc".Doca4);
END_REGION

REGION Network 8: Adaptação Tecnica
   RUNG wire#powerrail
      Move(in := "DB106_DadosEcuLine"."AGV.MAINLINE".ANDON, out1 => "DB211_DadosScada".Ecu.Andon)
   END_RUNG
   // the same network as SCL:
   "DB211_DadosScada".Ecu.Andon := "DB106_DadosEcuLine"."AGV.MAINLINE".ANDON;
END_REGION

REGION Network 9: Bloco de comunicação com os escravos
   // Este bloco realiza a escrita dos dados nos escravos da rede
   RUNG wire#powerrail
      "DB107_EnviaDados_DB"()
   END_RUNG
   // the same network as SCL:
   "DB107_EnviaDados_DB"();   // "FB107_EnviaDados"
END_REGION

REGION Network 10: Verifica o dia da semana esta programado para rodar o takt
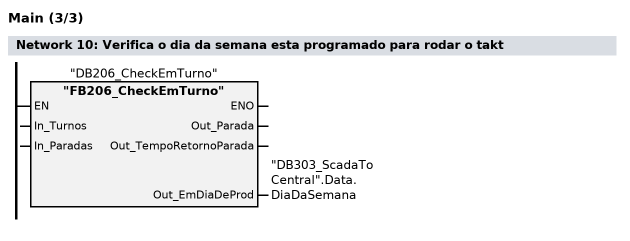
   RUNG wire#powerrail
      "DB206_CheckEmTurno"(In_Turnos :=, In_Paradas :=, Out_Parada =>, Out_TempoRetornoParada =>, Out_EmDiaDeProd => "DB303_ScadaToCentral".Data.DiaDaSemana)
   END_RUNG
   // the same network as SCL:
   "DB206_CheckEmTurno"(Out_EmDiaDeProd => "DB303_ScadaToCentral".Data.DiaDaSemana);   // "FB206_CheckEmTurno"
END_REGION
END_ORGANIZATION_BLOCK

// folder: 01_Comunicacao/01_FB

FUNCTION_BLOCK "FB100_CentralAgv_Comunicacao"   // FB100, SCL
TITLE = FB100_CentralAgv_Comunicacao
{ S7_Optimized_Access := 'TRUE' }
AUTHOR : ssbjvq
VERSION : 0.1
// FB100_CentralAgv_Comunicacao
   VAR_OUTPUT
      "Stop Time" : Int;
      Andons : Byte;
      Takt : Int;
      Objectivo : Int;
      Atual : Int;
   END_VAR
   VAR
      GET_CentralData : GET;
      S_Byte : Array[0..9] of Byte;
      GET_DadosAgvs : GET;
      GET_DadosAgvs_1 : GET;
      PUT_DadosCentralAgvs : PUT;
      Clock_Regulavel_Instance : "FB400_Clock_Regulavel";
      Date_Time : Date_And_Time;
      "Date" : Date;
      "Time" : Time_Of_Day;
   END_VAR
   VAR_TEMP
      Err : Int;
   END_VAR
BEGIN


   #GET_DadosAgvs(REQ := "Clock_0.5Hz",
                  ID := 16#103,
                  ADDR_1 := P#DB301.DBX0.0 Byte 144,
                  RD_1 := P#DB301.DBX0.0 Byte 144);

    #GET_DadosAgvs_1(REQ := NOT "Clock_0.5Hz" ,
                    ID := 16#103,
                    ADDR_1 := P#DB301.DBX144.0 Byte 144,
                    RD_1 := P#DB301.DBX144.0 Byte 144); 

   #GET_CentralData(REQ := "Clock_10Hz",
                    ID := 16#103,
                    ADDR_1 := P#DB301.DBX200.0 Byte 130,
                    RD_1 := P#DB301.DBX200.0 Byte 130); 



   REGION VerificaData
       #Clock_Regulavel_Instance(In_Tempo := T#20s);
       #Err := RD_SYS_T(#Date_Time);
       #Date := DTL_TO_DATE(#Date_Time);
       #Time := DTL_TO_TOD(#Date_Time);


       #PUT_DadosCentralAgvs(REQ := #Clock_Regulavel_Instance.Out_Pulso,
                             ID := 16#103,
                             ADDR_1 := P#DB300.DBX0.0 Byte 88,
                             SD_1 := P#DB303.DBX0.0 Byte 88);


      (* IF #Date = DTL_TO_DATE("DB302_InputDados".Ecu.Turnos."1_Turno".Inicio) THEN
           "DB303_ScadaToCentral".Data.Paradas_Programadas.Inicio[1] := "DB302_InputDados".Ecu.Paradas_Programadas_1Turno.Parada_2.Inicio;
           "DB303_ScadaToCentral".Data.Paradas_Programadas.Fim[1] := "DB302_InputDados".Ecu.Paradas_Programadas_1Turno.Parada_2.Fim;

           "DB303_ScadaToCentral".Data.Turnos.Inicio[0] := DTL_TO_TOD("DB302_InputDados".Ecu.Turnos."1_Turno".Inicio);
           "DB303_ScadaToCentral".Data.Turnos.Fim[0] := DTL_TO_TOD("DB302_InputDados".Ecu.Turnos."1_Turno".Fim);

       END_IF; *)

   END_REGION













   #Takt := DINT_TO_INT("DB301_CentralToScada".Data.Dados_Takt.Tempo_Takt);
   #"Stop Time" := DINT_TO_INT("DB301_CentralToScada".Data.Dados_Takt.Tempo_StopTime);
   #Objectivo := "DB301_CentralToScada".Data.Dados_Takt.Objetivo;
   #Atual := "DB301_CentralToScada".Data.Dados_Takt.Atual;
   //#Andons := ((BOOL_TO_BYTE("DB301_CentralToScada".Data.Dados_Takt.Andons[8]))+ (0+BOOL_TO_BYTE("DB301_CentralToScada".Data.Dados_Takt.Andons[7])+000000)+ BOOL_TO_BYTE("DB301_CentralToScada".Data.Dados_Takt.Andons[6])+ BOOL_TO_BYTE("DB301_CentralToScada".Data.Dados_Takt.Andons[5])+ BOOL_TO_BYTE("DB301_CentralToScada".Data.Dados_Takt.Andons[4])+ BOOL_TO_BYTE("DB301_CentralToScada".Data.Dados_Takt.Andons[3])+ BOOL_TO_BYTE("DB301_CentralToScada".Data.Dados_Takt.Andons[2])+ BOOL_TO_BYTE("DB301_CentralToScada".Data.Dados_Takt.Andons[1])+ BOOL_TO_BYTE("DB301_CentralToScada".Data.Dados_Takt.Andons[0]));
   #Andons := #S_Byte[9];


   IF "DB301_CentralToScada".Data.Dados_Takt.Andons[0] THEN
       #S_Byte[0] := 1;
   ELSE
       #S_Byte[0] := 0;
   END_IF;

   IF "DB301_CentralToScada".Data.Dados_Takt.Andons[1] THEN
       #S_Byte[1] := 2;
   ELSE
       #S_Byte[1] := 0;
   END_IF;

   IF "DB301_CentralToScada".Data.Dados_Takt.Andons[2] THEN
       #S_Byte[2] := 4;
   ELSE
       #S_Byte[2] := 0;
   END_IF;
   IF "DB301_CentralToScada".Data.Dados_Takt.Andons[3] THEN
       #S_Byte[3] := 8;
   ELSE
       #S_Byte[3] := 0;
   END_IF;
   IF "DB301_CentralToScada".Data.Dados_Takt.Andons[4] THEN
       #S_Byte[4] := 16;
   ELSE
       #S_Byte[4] := 0;
   END_IF;
   IF "DB301_CentralToScada".Data.Dados_Takt.Andons[5] THEN
       #S_Byte[5] := 32;
   ELSE
       #S_Byte[5] := 0;
   END_IF;
   IF "DB301_CentralToScada".Data.Dados_Takt.Andons[6] THEN
       #S_Byte[6] := 64;
   ELSE
       #S_Byte[6] := 0;
   END_IF;
   IF "DB301_CentralToScada".Data.Dados_Takt.Andons[7] THEN
       #S_Byte[7] := 128;
   ELSE
       #S_Byte[7] := 0;
   END_IF;
   IF "DB301_CentralToScada".Data.Dados_Takt.Andons[8] THEN
       #S_Byte[8] := 256;
   ELSE
       #S_Byte[8] := 0;
   END_IF;



   #S_Byte[9] := #S_Byte[8] + #S_Byte[7] + #S_Byte[6] + #S_Byte[5] + #S_Byte[4] + #S_Byte[3] + #S_Byte[2] + #S_Byte[1] + #S_Byte[0];
END_FUNCTION_BLOCK

FUNCTION_BLOCK "FB101_ComunicacaoEscravos"   // FB101, LAD
{ S7_Optimized_Access := 'TRUE' }
VERSION : 0.1
// Este bloco centraliza a leitura dos dados das linhas
   VAR
      GetCabLine : "FB102_GetInformation";
      GetSKDLine : "FB102_GetInformation";
      GetSkidLine : "FB102_GetInformation";
   END_VAR
BEGIN

REGION Network 1: Cab Line
   // Realiza a leitura das informações da linha de Cabinas
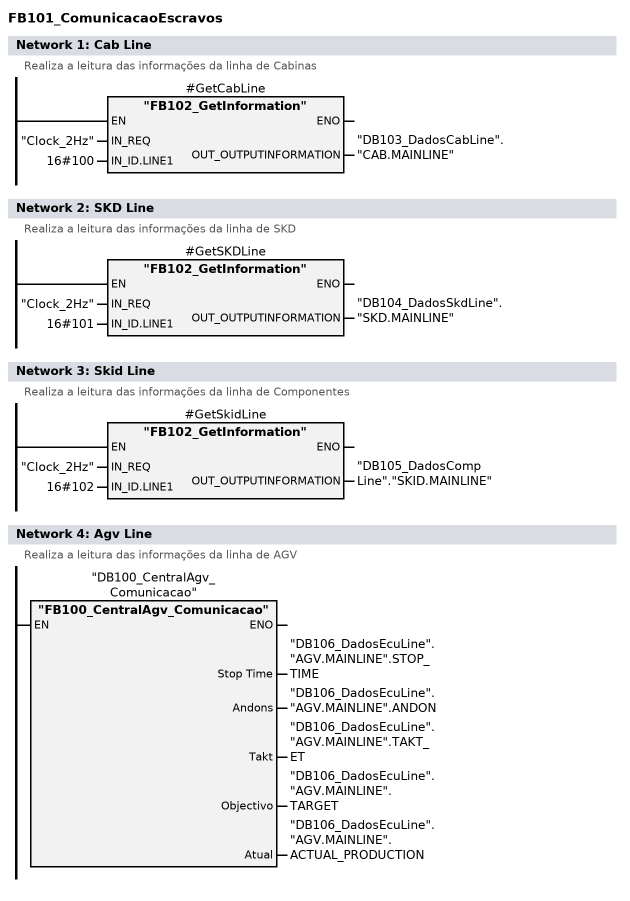
   RUNG wire#powerrail
      #GetCabLine(IN_REQ := "Clock_2Hz", "IN_ID.LINE1" := 16#100, OUT_OUTPUTINFORMATION => "DB103_DadosCabLine"."CAB.MAINLINE")
   END_RUNG
   // the same network as SCL:
   #GetCabLine(IN_REQ := "Clock_2Hz",   // "FB102_GetInformation"
               "IN_ID.LINE1" := 16#100,
               OUT_OUTPUTINFORMATION => "DB103_DadosCabLine"."CAB.MAINLINE");
END_REGION

REGION Network 2: SKD Line
   // Realiza a leitura das informações da linha de SKD
   RUNG wire#powerrail
      #GetSKDLine(IN_REQ := "Clock_2Hz", "IN_ID.LINE1" := 16#101, OUT_OUTPUTINFORMATION => "DB104_DadosSkdLine"."SKD.MAINLINE")
   END_RUNG
   // the same network as SCL:
   #GetSKDLine(IN_REQ := "Clock_2Hz",   // "FB102_GetInformation"
               "IN_ID.LINE1" := 16#101,
               OUT_OUTPUTINFORMATION => "DB104_DadosSkdLine"."SKD.MAINLINE");
END_REGION

REGION Network 3: Skid Line
   // Realiza a leitura das informações da linha de Componentes
   RUNG wire#powerrail
      #GetSkidLine(IN_REQ := "Clock_2Hz", "IN_ID.LINE1" := 16#102, OUT_OUTPUTINFORMATION => "DB105_DadosCompLine"."SKID.MAINLINE")
   END_RUNG
   // the same network as SCL:
   #GetSkidLine(IN_REQ := "Clock_2Hz",   // "FB102_GetInformation"
                "IN_ID.LINE1" := 16#102,
                OUT_OUTPUTINFORMATION => "DB105_DadosCompLine"."SKID.MAINLINE");
END_REGION

REGION Network 4: Agv Line
   // Realiza a leitura das informações da linha de AGV
   RUNG wire#powerrail
      "DB100_CentralAgv_Comunicacao"("Stop Time" => "DB106_DadosEcuLine"."AGV.MAINLINE".STOP_TIME, Andons => "DB106_DadosEcuLine"."AGV.MAINLINE".ANDON, Takt => "DB106_DadosEcuLine"."AGV.MAINLINE".TAKT_ET, Objectivo => "DB106_DadosEcuLine"."AGV.MAINLINE".TARGET, Atual => "DB106_DadosEcuLine"."AGV.MAINLINE".ACTUAL_PRODUCTION)
   END_RUNG
   // the same network as SCL:
   "DB100_CentralAgv_Comunicacao"("Stop Time" => "DB106_DadosEcuLine"."AGV.MAINLINE".STOP_TIME,   // "FB100_CentralAgv_Comunicacao"
                           Andons => "DB106_DadosEcuLine"."AGV.MAINLINE".ANDON,
                           Takt => "DB106_DadosEcuLine"."AGV.MAINLINE".TAKT_ET,
                           Objectivo => "DB106_DadosEcuLine"."AGV.MAINLINE".TARGET,
                           Atual => "DB106_DadosEcuLine"."AGV.MAINLINE".ACTUAL_PRODUCTION);
END_REGION
END_FUNCTION_BLOCK

FUNCTION_BLOCK "FB102_GetInformation"   // FB102, SCL
{ S7_Optimized_Access := 'TRUE' }
VERSION : 0.1
   VAR_INPUT
      IN_REQ : Bool;
      "IN_ID.LINE1" : Word;
   END_VAR
   VAR_OUTPUT
      OUT_OUTPUTINFORMATION : "TAKT_OUTPUT.INFORMATION";
   END_VAR
   VAR
      "GET_TAKT.LINE1" : GET;
      "S_REQ.TAKT.LINE1" : Bool;
      "S_ID.TAKT.LINE1" : Word;
      "S_NDR.TAKT.LINE1" : Bool;
      "S_ERROR.TAKT.LINE1" : Bool;
      "S_STATUS.TAKT.LINE1" : Word;
      "S_RD_1.TAKT.LINE1" : Int;
      "S_RD_2.STOP.LINE1" : Int;
      "S_RD_3.ACTUAL.LINE1" : Int;
      "S_RD_4.TARGET.LINE1" : Int;
      "GET_ANDON.LINE1" : GET;
      "S_REQ.ANDON.LINE1" : Bool;
      "S_ID.ANDON.LINE1" : Word;
      "S_NDR.ANDON.LINE1" : Bool;
      "S_ERROR.ANDON.LINE1" : Bool;
      "S_STATUS.ANDON.LINE1" : Word;
      "S_RD_1.ANDON.LINE1" : Byte;
   END_VAR
BEGIN
   (*GET INFORMATION FROM LINE 1 - CAB*)

   //READ INPUT
   #"S_REQ.TAKT.LINE1" := #IN_REQ;
   #"S_ID.TAKT.LINE1" := #"IN_ID.LINE1";
   #"S_REQ.ANDON.LINE1" := #IN_REQ;
   #"S_ID.ANDON.LINE1" := #"IN_ID.LINE1";

   //GET TAKT TIME
   #"GET_TAKT.LINE1"(REQ := #"S_REQ.TAKT.LINE1",
             ID := #"S_ID.TAKT.LINE1",
             ADDR_1 := P#DB23.DBX0.0 BYTE 2, //TAKT
             ADDR_2 := P#DB23.DBX6.0 BYTE 2, //STOP
             ADDR_3 := P#DB23.DBX4.0 BYTE 2, //ACTUAL
             ADDR_4 := P#DB23.DBX8.0 BYTE 2, //TARGET
             RD_1 := #"S_RD_1.TAKT.LINE1",
             RD_2 := #"S_RD_2.STOP.LINE1",
             RD_3 := #"S_RD_3.ACTUAL.LINE1",
             RD_4 := #"S_RD_4.TARGET.LINE1",
             ERROR => #"S_ERROR.TAKT.LINE1",
             NDR => #"S_NDR.TAKT.LINE1",
             STATUS => #"S_STATUS.TAKT.LINE1");

   //GET ANDON SIGNAL
   #"GET_ANDON.LINE1" (REQ := #"S_REQ.ANDON.LINE1",
               ID := #"S_ID.ANDON.LINE1",
               ADDR_1 := P#DB23.DBX2.0 BYTE 1,
               RD_1 := #"S_RD_1.ANDON.LINE1",
               ERROR => #"S_ERROR.ANDON.LINE1",
               NDR => #"S_NDR.ANDON.LINE1",
               STATUS =>#"S_STATUS.ANDON.LINE1");

   //WRITE OUTPUT
   #OUT_OUTPUTINFORMATION.TAKT_ET:= #"S_RD_1.TAKT.LINE1";
   #OUT_OUTPUTINFORMATION.STOP_TIME := #"S_RD_2.STOP.LINE1";
   #OUT_OUTPUTINFORMATION.ACTUAL_PRODUCTION := #"S_RD_3.ACTUAL.LINE1";
   #OUT_OUTPUTINFORMATION.TARGET := #"S_RD_4.TARGET.LINE1";
   #OUT_OUTPUTINFORMATION."ANDON" := #"S_RD_1.ANDON.LINE1";

   //------------------------------------------------------------------------------------------------------------------------------------------------------------------------------------\\
END_FUNCTION_BLOCK

FUNCTION_BLOCK "FB107_EnviaDados"   // FB107, SCL
TITLE = FB107_EnviaDados
{ S7_Optimized_Access := 'TRUE' }
VERSION : 0.1
   VAR RETAIN
      "Counter" : CTU_INT;
   END_VAR
   VAR
      PUT_PowertrainEcu : PUT;
      PUT_PowertrainEcu_1 : PUT;
      PUT_PowertrainEcu_2 : PUT;
      PUT_PowertrainEcu_3 : PUT;
      PUT_Cabinas : PUT;
      PUT_Skd : PUT;
      PUT_Componentes : PUT;
      Clock_Regulavel : "FB400_Clock_Regulavel";
      S_Array : Array[0..20] of Bool;
      S_Sinal : Bool;
   END_VAR
BEGIN

   REGION LogicaDeChamadaDePUT
       #Clock_Regulavel(In_Tempo := T#60s,
                        Out_Sinal => #S_Sinal);

       #Counter(CU := #S_Sinal,
                R := #S_Array[7],
                PV := 5);


       CASE #Counter.CV OF
           0:
               #S_Array[7] := 0;
               #S_Array[0] := 1;
           1:
               #S_Array[0] := 0;
               #S_Array[1] := 1;
           2:
               #S_Array[1] := 0;
               #S_Array[2] := 1;
           3:
               #S_Array[2] := 0;
               #S_Array[3] := 1;
           4:
               #S_Array[3] := 0;
               #S_Array[4] := 1;
           5: // Reset contador
               #S_Array[4] := 0;
               #S_Array[5] := 1;
           6:
               #S_Array[5] := 0;
               #S_Array[6] := 1;
           7:
               #S_Array[6] := 0;
               #S_Array[7] := 1;
           ELSE
               #S_Array[0] := 0;
               #S_Array[1] := 0;
               #S_Array[2] := 0;
               #S_Array[3] := 0;
               #S_Array[4] := 0;
       END_CASE;

   END_REGION



   REGION BlocosPUT
       #PUT_Cabinas(REQ := #S_Array[0],
                    ID := 16#100,
                    ADDR_1 := P#DB500.DBX0.0 BYTE 500,//Partner
                    SD_1 := P#DB214.DBX0.0 BYTE 500);//Local

       #PUT_Skd(REQ := #S_Array[1],
                ID := 16#101,
                ADDR_1 := P#DB500.DBX0.0 BYTE 500,//Partner
                SD_1 := P#DB214.DBX504.0 BYTE 500);//Local

       #PUT_Componentes(REQ := #S_Array[2],
                        ID := 16#102,
                        ADDR_1 := P#DB500.DBX0.0 BYTE 500,//Partner
                        SD_1 := P#DB214.DBX1008.0 BYTE 500);//Local
       REGION PowertrainEcu
           #PUT_PowertrainEcu(REQ := #S_Array[3],
                              ID := 16#103,
                              ADDR_1 := P#DB500.DBX0.0 BYTE 144,//Partner
                              SD_1 := P#DB214.DBX1512.0 BYTE 144);//Local
           #PUT_PowertrainEcu_1(REQ := #S_Array[4],
                                ID := 16#103,
                                ADDR_1 := P#DB500.DBX144.0 BYTE 144,//Partner
                                SD_1 := P#DB214.DBX1656.0 BYTE 144);//Local 
           #PUT_PowertrainEcu_2(REQ := #S_Array[5],
                                ID := 16#103,
                                ADDR_1 := P#DB500.DBX288.0 BYTE 144,//Partner
                                SD_1 := P#DB214.DBX1800.0 BYTE 144);//Local 
           #PUT_PowertrainEcu_3(REQ := #S_Array[6],
                                ID := 16#103,
                                ADDR_1 := P#DB500.DBX432.0 BYTE 68,//Partner
                                SD_1 := P#DB214.DBX1944.0 BYTE 68);//Local 
       END_REGION


   END_REGION
END_FUNCTION_BLOCK

// folder: 02_Takt/01_FB

FUNCTION_BLOCK "FB200_FiltroDados_Cab"   // FB200, SCL
TITLE = FB200_FiltroDadosTakt
{ S7_Optimized_Access := 'TRUE' }
VERSION : 0.1
// Realiza o filtro das infos e sobe e coloca na DB 1000
   VAR_INPUT
      In_InfoCabinas : "TAKT_OUTPUT.INFORMATION";
      In_Turno : Struct
         Turnos : Array[0..2] of Struct
            Inicio : Date_And_Time;
            Fim : Date_And_Time;
            Objetivo : Int;
            DiasDaSemana : Array[0..6] of Bool;
            Paradas : Array[0..5] of Struct
               Inicio : Date_And_Time;
               Fim : Date_And_Time;
            END_STRUCT;
            HE_Inicio : Date_And_Time;
            HE_Fim : Date_And_Time;
         END_STRUCT;
      END_STRUCT;
   END_VAR
   VAR_OUTPUT
      Out_Linha : Struct
         Tempo_Takt : DInt;
         Tempo_StopTime : DInt;
         Objetivo : Int;
         Atual : Int;
         LinhaParada : Bool;
         TempoRetornoParada : DInt;
         LinhaRodando : Bool;
         Andons : Array[0..8] of Bool;
         CorDeTela : Byte;
         DirectRun : Real;
         SaldoDoTurno : Int;
         AndonOn : Int;
         Paradas : Array[0..1] of Struct
            Inicio : Time_Of_Day;
            Fim : Time_Of_Day;
            Posto : Int;
            ValorTimer : Int;
            ValorTimerFim : Int;
         END_STRUCT;
         NumMensagem : Int;
         Emergencias : Array[0..8] of Bool;
      END_STRUCT;
      Out_Mensagem : String;
   END_VAR
   VAR
      S_DateTime : Date_And_Time;
      S_CounterFor : Int;
      S_CounterFor_1 : Int;
      S_Turnos : Array[0..2] of Struct
         Paradas : Array[0..6] of Bool;
         ContagemRetorno : Array[0..6] of DInt;
      END_STRUCT;
      S_ForaDeTurno : Bool;
      S_TempoRetorno : DInt;
      S_Hora : Time_Of_Day;
   END_VAR
   VAR_TEMP
      Err : Int;
   END_VAR
BEGIN
   (*
       ESTE BLOCO REALIZA O FILTRO DAS INFORMAÇÕES DO TAKT, EXEMPLOS: TROCA DA COR DA TELA, MENSAGENS NA TELA E ETC
   *)


   // Converte o sinal de andon de byte para boolean
   REGION Valores ANDON
       // Converte o sinal de andon de byte para boolean
       #Out_Linha.Andons[0] := #In_InfoCabinas.ANDON.%X0;
       #Out_Linha.Andons[1] := #In_InfoCabinas.ANDON.%X1;
       #Out_Linha.Andons[2] := #In_InfoCabinas.ANDON.%X2;
       #Out_Linha.Andons[3] := #In_InfoCabinas.ANDON.%X3;
       #Out_Linha.Andons[4] := #In_InfoCabinas.ANDON.%X4;
       #Out_Linha.Andons[5] := #In_InfoCabinas.ANDON.%X5;
       #Out_Linha.Andons[6] := #In_InfoCabinas.ANDON.%X6;
       #Out_Linha.Andons[7] := #In_InfoCabinas.ANDON.%X7;
   END_REGION

   // Converte o sinal de emergencia de byte para boolean
   REGION Valores Emergencia
       // Converte o sinal de emergencia de byte para boolean
       #Out_Linha.Emergencias[0] := #In_InfoCabinas.EMERGENCY.%X0;
       #Out_Linha.Emergencias[1] := #In_InfoCabinas.EMERGENCY.%X1;
       #Out_Linha.Emergencias[2] := #In_InfoCabinas.EMERGENCY.%X2;
       #Out_Linha.Emergencias[3] := #In_InfoCabinas.EMERGENCY.%X3;
       #Out_Linha.Emergencias[4] := #In_InfoCabinas.EMERGENCY.%X4;
       #Out_Linha.Emergencias[5] := #In_InfoCabinas.EMERGENCY.%X5;
       #Out_Linha.Emergencias[6] := #In_InfoCabinas.EMERGENCY.%X6;
       #Out_Linha.Emergencias[7] := #In_InfoCabinas.EMERGENCY.%X7;
   END_REGION

   //Realiza a leitura da hora atual do CLP
   REGION HoraAtual

       //Realiza a leitura da hora atual do CLP
       #Err := RD_LOC_T(#S_DateTime);

   END_REGION
   REGION VerificaEmTurno
       #S_Hora := DT_TO_TOD(#S_DateTime);
       IF #S_Hora > TOD#16:00:00 THEN
           #S_TempoRetorno := TOD_TO_DINT(TOD#07:00:00) - TOD_TO_DINT(#S_Hora);
           #S_ForaDeTurno := 1;
       ELSE
           #S_TempoRetorno := 0;
           #S_ForaDeTurno := 0;
       END_IF;


   END_REGION
   //Verifica se a linha esta em turno, caso não esteja retorno o tempo necessario para a linha voltar a rodar
   REGION LinhaEmTurno
       FOR #S_CounterFor := 0 TO 2 DO
           //Verifica se está em turno
           IF #In_Turno.Turnos[#S_CounterFor].Inicio >= #S_DateTime AND #S_DateTime <= #In_Turno.Turnos[#S_CounterFor].Fim THEN
               //Verifica se existe alguma parada programada
               FOR #S_CounterFor_1 := 0 TO 5 DO
                   IF #In_Turno.Turnos[#S_CounterFor].Paradas[#S_CounterFor_1].Inicio >= #S_DateTime
                       AND #S_DateTime <= #In_Turno.Turnos[#S_CounterFor].Paradas[#S_CounterFor_1].Fim THEN

                       #S_Turnos[#S_CounterFor].Paradas[#S_CounterFor_1] := 1;
                       #S_Turnos[#S_CounterFor].ContagemRetorno[#S_CounterFor_1] := TOD_TO_DINT(DT_TO_TOD(#S_DateTime - (#In_Turno.Turnos[#S_CounterFor].Paradas[#S_CounterFor_1].Fim - #In_Turno.Turnos[#S_CounterFor].Paradas[#S_CounterFor_1].Inicio)));
                   ELSE
                       #S_Turnos[#S_CounterFor].ContagemRetorno[#S_CounterFor_1] := 0;
                       #S_Turnos[#S_CounterFor].Paradas[#S_CounterFor_1] := 0;

                   END_IF;

                   #S_Turnos[#S_CounterFor].Paradas[6] := 0; // Em turno
                   #S_Turnos[#S_CounterFor].ContagemRetorno[6] := 0;
               END_FOR;
           ELSE
               #S_Turnos[#S_CounterFor].Paradas[6] := 1; // Fora de turno
               #S_Turnos[#S_CounterFor].ContagemRetorno[6] := #S_DateTime - #In_Turno.Turnos[#S_CounterFor].Paradas[#S_CounterFor_1].Inicio; // Quantidade de tempo restante para reiniciar o novo turno
           END_IF;

       END_FOR;

       #S_ForaDeTurno := #S_Turnos[0 AND 1 AND 2].Paradas[0 AND 1 AND 2 AND 3 AND 4 AND 5 AND 6];
       #S_TempoRetorno := #S_Turnos[0 AND 1 AND 2].ContagemRetorno[0 AND 1 AND 2 AND 3 AND 4 AND 5 AND 6];
   END_REGION

   // Realiza a analise de todos os dados e troca a cor da tela
   REGION DefiniçãoCorDaTela
       // 1 - Tela Amarela (Necessario ajuda em algum posto e não estourou o tempo do TAKT)
       IF ((#Out_Linha.Andons[1] OR #Out_Linha.Andons[2] OR #Out_Linha.Andons[3] OR #Out_Linha.Andons[4] OR #Out_Linha.Andons[5]) AND (#In_InfoCabinas.TAKT_ET > 0)) AND NOT #S_ForaDeTurno THEN
           #Out_Linha.CorDeTela := 1;

       // 2 - Tela Vermelho (Necessario ajuda em algum posto e estourou o tempo do TAKT)
       ELSIF (((#Out_Linha.Andons[1] OR #Out_Linha.Andons[2] OR #Out_Linha.Andons[3] OR #Out_Linha.Andons[4] OR #Out_Linha.Andons[5]) AND (#In_InfoCabinas.TAKT_ET <= 0)) OR (#In_InfoCabinas.EMERGENCY <> 0)) AND NOT #S_ForaDeTurno THEN
           #Out_Linha.CorDeTela := 2;

       //3 - Tela Azul - (Aguardando inicio de turno/Volta da refeição)
       ELSIF #S_ForaDeTurno THEN
           #Out_Linha.CorDeTela := 3;

       //4 - Tela Laranja - (Aguardando retirada do produto)
       ELSIF ((#Out_Linha.Andons[7]) OR #Out_Linha.Andons[7]) AND NOT #S_ForaDeTurno  THEN
           #Out_Linha.CorDeTela := 4;
       //0 - Tela Branca/Preta (Tudo Ok)
       ELSE
           #Out_Linha.CorDeTela := 0;
       END_IF;


   END_REGION

   // Realiza a analise de todos os dados e escreve a mensagem na tela 
   REGION Mensagens

       IF #In_InfoCabinas.EMERGENCY <> 0 AND NOT #S_ForaDeTurno THEN

               // Sinal de EMERGÊNCIA  do posto 1
           IF #Out_Linha.Emergencias[0] THEN
               #Out_Linha.NumMensagem := 1;
               #Out_Mensagem := 'EMERGÊNCIA  ACIONADO NO POSTO 1';

               // Sinal de EMERGÊNCIA  do posto 2
           ELSIF #Out_Linha.Emergencias[1] THEN
               #Out_Linha.NumMensagem := 2;
               #Out_Mensagem := 'EMERGÊNCIA  ACIONADO NO POSTO 2';

               // Sinal de EMERGÊNCIA  do posto 3
           ELSIF #Out_Linha.Emergencias[2] THEN
               #Out_Linha.NumMensagem := 3;
               #Out_Mensagem := 'EMERGÊNCIA  ACIONADO NO POSTO 3';

               // Sinal de EMERGÊNCIA  do posto 4
           ELSIF #Out_Linha.Emergencias[3] THEN
               #Out_Linha.NumMensagem := 4;
               #Out_Mensagem := 'EMERGÊNCIA  ACIONADO NO POSTO 4';

               // Sinal de EMERGÊNCIA  do posto 5
           ELSIF #Out_Linha.Emergencias[4] THEN
               #Out_Linha.NumMensagem := 5;
               #Out_Mensagem := 'EMERGÊNCIA  ACIONADO NO POSTO 5';

               // Sinal de EMERGÊNCIA  do posto 6
           ELSIF #Out_Linha.Emergencias[5] THEN
               #Out_Linha.NumMensagem := 6;
               #Out_Mensagem := 'EMERGÊNCIA  ACIONADO NO POSTO 6';

               // Sinal de EMERGÊNCIA  do posto 7
           ELSIF #Out_Linha.Emergencias[6] THEN
               #Out_Linha.NumMensagem := 7;
               #Out_Mensagem := 'EMERGÊNCIA  ACIONADO NO POSTO 7';

               // Sinal de EMERGÊNCIA  do posto 8
           ELSIF #Out_Linha.Emergencias[7] THEN
               #Out_Linha.NumMensagem := 8;
               #Out_Mensagem := 'EMERGÊNCIA  ACIONADO NO POSTO 8';

           END_IF;

       ELSIF #In_InfoCabinas.ANDON <> 0 AND NOT #S_ForaDeTurno THEN

               // Sinal de andon do posto 1
           IF #Out_Linha.Andons[0] THEN
               #Out_Linha.NumMensagem := 9;
               #Out_Mensagem := 'TROCADOR DE SKID EM PROCESSO';

               // Sinal de andon do posto 2
           ELSIF #Out_Linha.Andons[1] THEN
               #Out_Linha.NumMensagem := 10;
               #Out_Mensagem := 'NECESSARIO AJUDA NO POSTO 2';

               // Sinal de andon do posto 3
           ELSIF #Out_Linha.Andons[2] THEN
               #Out_Linha.NumMensagem := 11;
               #Out_Mensagem := 'NECESSARIO AJUDA NO POSTO 3';

               // Sinal de andon do posto 4
           ELSIF #Out_Linha.Andons[3] THEN
               #Out_Linha.NumMensagem := 12;
               #Out_Mensagem := 'NECESSARIO AJUDA NO POSTO 4';

               // Sinal de andon do posto 5
           ELSIF #Out_Linha.Andons[4] THEN
               #Out_Linha.NumMensagem := 13;
               #Out_Mensagem := 'NECESSARIO AJUDA NO POSTO 5';

               // Sinal de andon do posto 6
           ELSIF #Out_Linha.Andons[5] THEN
               #Out_Linha.NumMensagem := 14;
               #Out_Mensagem := 'NECESSARIO AJUDA NO POSTO 6';

               // Sinal de andon do posto 7
           ELSIF #Out_Linha.Andons[6] THEN
               #Out_Linha.NumMensagem := 15;
               #Out_Mensagem := 'QUALITY GATE INSPECIONANDO O PRODUTO POSTO 7';

               // Sinal de andon do posto 8
           ELSIF #Out_Linha.Andons[7] THEN
               #Out_Linha.NumMensagem := 16;
               #Out_Mensagem := 'AGUARDANDO RETIRADA DO PRODUTO NO POSTO 8';

           END_IF;
           ;
           // Linha em parada de produção
       ELSIF #S_ForaDeTurno THEN
           #Out_Linha.NumMensagem := 17;
           #Out_Mensagem := 'LINHA EM PARADA DE PRODUÇÃO';
       ELSE
           #Out_Linha.NumMensagem := 0;
           #Out_Mensagem := 'LINHA LIBERADA';
       END_IF;

   END_REGION

   // Coloca os dados das memorias nas saidas do bloco
   REGION Saidas
       // Coloca os dados das memorias nas saidas do bloco
       #Out_Linha.Tempo_Takt := #In_InfoCabinas.TAKT_ET;
       #Out_Linha.Tempo_StopTime := #In_InfoCabinas.STOP_TIME;
       #Out_Linha.Objetivo := #In_InfoCabinas.TARGET;
       #Out_Linha.Atual := #In_InfoCabinas.ACTUAL_PRODUCTION;
       #Out_Linha.DirectRun := 99.9;
       #Out_Linha.LinhaParada := #S_ForaDeTurno;
       #Out_Linha.TempoRetornoParada := #S_TempoRetorno;
       #Out_Linha.LinhaRodando := NOT #S_ForaDeTurno;
   END_REGION
END_FUNCTION_BLOCK

FUNCTION_BLOCK "FB201_FiltragemDados"   // FB201, SCL
TITLE = Filtragem de Dados dos Takts
{ S7_Optimized_Access := 'TRUE' }
VERSION : 0.1
   VAR_INPUT
      In_DadosCabinas : "TAKT_OUTPUT.INFORMATION";   // Dados da linha de Cabinas
      In_DadosSKD : "TAKT_OUTPUT.INFORMATION";   // Dados da linha de SKD
      In_DadosComp : "TAKT_OUTPUT.INFORMATION";   // Dados da linha de Componentes
      In_DadosEcu : "Central.Database";   // Dados da linha de Ecu
   END_VAR
   VAR_OUTPUT
      Out_LinhaCabinas : Struct
         Tempo_Takt : DInt;
         Tempo_StopTime : DInt;
         Objetivo : Int;
         Atual : Int;
         LinhaParada : Bool;
         TempoRetornoParada : DInt;
         LinhaRodando : Bool;
         Andons : Array[0..8] of Bool;
         CorDeTela : Byte;
         DirectRun : Real;
         SaldoDoTurno : Int;
         AndonOn : Int;
         Paradas : Array[0..1] of Struct
            Inicio : Time_Of_Day;
            Fim : Time_Of_Day;
            Posto : Int;
            ValorTimer : Int;
            ValorTimerFim : Int;
         END_STRUCT;
         NumMensagem : Int;
         Emergencias : Array[0..8] of Bool;
      END_STRUCT;
      Out_MensagemCab : String;
      Out_LinhaSkd : Struct
         Tempo_Takt : DInt;
         Tempo_StopTime : DInt;
         Objetivo : Int;
         Atual : Int;
         LinhaParada : Bool;
         TempoRetornoParada : DInt;
         LinhaRodando : Bool;
         Andons : Array[0..8] of Bool;
         CorDeTela : Byte;
         DirectRun : Real;
         SaldoDoTurno : Int;
         AndonOn : Int;
         Paradas : Array[0..1] of Struct
            Inicio : Time_Of_Day;
            Fim : Time_Of_Day;
            Posto : Int;
            ValorTimer : Int;
            ValorTimerFim : Int;
         END_STRUCT;
         NumMensagem : Int;
         Emergencias : Array[0..8] of Bool;
      END_STRUCT;
      Out_MensagemSkd : String;
      Out_LinhaComp : Struct
         Tempo_Takt : DInt;
         Tempo_StopTime : DInt;
         Objetivo : Int;
         Atual : Int;
         LinhaParada : Bool;
         TempoRetornoParada : DInt;
         LinhaRodando : Bool;
         Andons : Array[0..8] of Bool;
         CorDeTela : Byte;
         DirectRun : Real;
         SaldoDoTurno : Int;
         AndonOn : Int;
         Paradas : Array[0..1] of Struct
            Inicio : Time_Of_Day;
            Fim : Time_Of_Day;
            Posto : Int;
            ValorTimer : Int;
            ValorTimerFim : Int;
         END_STRUCT;
         NumMensagem : Int;
         Emergencias : Array[0..8] of Bool;
      END_STRUCT;
      Out_MensagemComp : String;
      Out_LinhaEcu : Struct
         Tempo_Takt : DInt;
         Tempo_StopTime : DInt;
         Objetivo : Int;
         Atual : Int;
         LinhaParada : Bool;
         TempoRetornoParada : DInt;
         LinhaRodando : Bool;
         Andons : Array[0..8] of Bool;
         CorDeTela : Byte;
         DirectRun : Real;
         SaldoDoTurno : Int;
         AndonOn : Int;
         Paradas : Array[0..1] of Struct
            Inicio : Time_Of_Day;
            Fim : Time_Of_Day;
            Posto : Int;
            ValorTimer : Int;
            ValorTimerFim : Int;
         END_STRUCT;
         NumMensagem : Int;
         Emergencias : Array[0..8] of Bool;
      END_STRUCT;
      Out_MensagemEcu : String;
      Out_DadosTakt : "DadosDosTakts";
   END_VAR
   VAR
      FiltroDadosTakt_Cabinas : "FB200_FiltroDados_Cab";
      FiltroDadosTakt_Skd : "FB203_FiltroDados_Skd";
      FiltroDadosTakt_Comp : "FB204_FiltroDados_Comp";
      FiltroDados_TaktAgvs : "FB202_FiltroDados_TaktAgvs";
      FiltroDadosAgv : Array[0..9] of "FB205_FiltroDadosAgv";
   END_VAR
BEGIN


   // Realiza o filtro dos dados por linha e formata no padrão que o sistema deve receber
   REGION FiltrosPorLinha
       // Filtro da linha de cabinas
       #FiltroDadosTakt_Cabinas(In_InfoCabinas := #In_DadosCabinas,
                                (* In_Turno := #In_DadosTurnos.Linha_Cabinas, *)
                                Out_Linha => #Out_LinhaCabinas,
                                Out_Mensagem => #Out_MensagemCab);
       // Filtro da linha de SKD
       #FiltroDadosTakt_Skd(In_InfoCabinas := #In_DadosSKD,
                            (* In_Turno := #In_DadosTurnos.Linha_SKD, *)
                            Out_Linha => #Out_LinhaSkd,
                            Out_Mensagem => #Out_MensagemSkd);

       // Filtro da linha de Componentes
       #FiltroDadosTakt_Comp(In_InfoCabinas := #In_DadosComp,
                           (* In_Turno := #In_DadosTurnos.Linha_Componentes, *)
                            Out_Linha => #Out_LinhaComp,
                            Out_Mensagem => #Out_MensagemComp);

      // Filtro da linha de ECU -  (*  Diferente dos outros blocos, por conta dos AGVs  *)
      #FiltroDados_TaktAgvs(In_DadosEcu:=#In_DadosEcu,
                            (* In_Turno:=#In_DadosTurnos.Linha_ECU, *)
                            Out_LinhaEcu=>#Out_LinhaEcu,
                            Out_MensagemEcu=>#Out_MensagemEcu);

   END_REGION

   //Formata os dados no modelo que a IHM usa.
   REGION FormatadorDadosTakt
       #Out_DadosTakt.Linhas_Cabinas := #Out_LinhaCabinas;
       #Out_DadosTakt.Mensagem_Cab := #Out_MensagemCab;
       #Out_DadosTakt.Linhas_SKD := #Out_LinhaSkd;
       #Out_DadosTakt.Mensagem_Skd := #Out_MensagemSkd;
       #Out_DadosTakt.Linhas_EixoMotor := #Out_LinhaComp;
       #Out_DadosTakt.Mensagem_Comp := #Out_MensagemComp ;
       #Out_DadosTakt.Linhas_ECU := #Out_LinhaEcu;
       #Out_DadosTakt.Mensagem_Ecu := #Out_MensagemEcu;
   END_REGION


   //Formata os dados no modelo que a Sistema                    usa.
   REGION FormatadorDadosTakt2
       "DB211_DadosScada".Cabinas.Timer := DINT_TO_INT(#Out_LinhaCabinas.Tempo_Takt);
       "DB211_DadosScada".Cabinas.StopTime := DINT_TO_INT(#Out_LinhaCabinas.Tempo_StopTime);
       "DB211_DadosScada".Cabinas.Objetivo := INT_TO_BYTE(#Out_LinhaCabinas.Objetivo);
       "DB211_DadosScada".Cabinas.Atual := INT_TO_BYTE(#Out_LinhaCabinas.Atual);
       "DB211_DadosScada".Cabinas.TempoRetornoParada := DINT_TO_INT(#Out_LinhaCabinas.TempoRetornoParada);
       "DB211_DadosScada".Cabinas.Andon := #In_DadosCabinas.ANDON;
       "DB211_DadosScada".Cabinas.Emergencia := #In_DadosCabinas.EMERGENCY;
       "DB211_DadosScada".Cabinas.CorDeTela := #Out_LinhaCabinas.CorDeTela;
       "DB211_DadosScada".Cabinas.NumMensagem := INT_TO_BYTE(#Out_LinhaCabinas.NumMensagem);

       "DB211_DadosScada".Skd.Timer := DINT_TO_INT(#Out_LinhaSkd.Tempo_Takt);
       "DB211_DadosScada".Skd.StopTime := DINT_TO_INT(#Out_LinhaSkd.Tempo_StopTime);
       "DB211_DadosScada".Skd.Objetivo := INT_TO_BYTE(#Out_LinhaSkd.Objetivo);
       "DB211_DadosScada".Skd.Atual := INT_TO_BYTE(#Out_LinhaSkd.Atual);
       "DB211_DadosScada".Skd.TempoRetornoParada := DINT_TO_INT(#Out_LinhaSkd.TempoRetornoParada);
       "DB211_DadosScada".Skd.Andon := #In_DadosSKD.ANDON;
       "DB211_DadosScada".Skd.Emergencia := #In_DadosSKD.EMERGENCY;
       "DB211_DadosScada".Skd.CorDeTela := #Out_LinhaSkd.CorDeTela;
       "DB211_DadosScada".Skd.NumMensagem := INT_TO_BYTE(#Out_LinhaSkd.NumMensagem);

       "DB211_DadosScada".Comp.Timer := DINT_TO_INT(#Out_LinhaComp.Tempo_Takt);
       "DB211_DadosScada".Comp.StopTime := DINT_TO_INT(#Out_LinhaComp.Tempo_StopTime);
       "DB211_DadosScada".Comp.Objetivo := INT_TO_BYTE(#Out_LinhaComp.Objetivo);
       "DB211_DadosScada".Comp.Atual := INT_TO_BYTE(#Out_LinhaComp.Atual);
       "DB211_DadosScada".Comp.TempoRetornoParada := DINT_TO_INT(#Out_LinhaComp.TempoRetornoParada);
       "DB211_DadosScada".Comp.Andon := #In_DadosComp.ANDON;
       "DB211_DadosScada".Comp.Emergencia := #In_DadosComp.EMERGENCY;
       "DB211_DadosScada".Comp.CorDeTela := #Out_LinhaComp.CorDeTela;
       "DB211_DadosScada".Comp.NumMensagem := INT_TO_BYTE(#Out_LinhaComp.NumMensagem);

       "DB211_DadosScada".Ecu.Timer := DINT_TO_INT(#Out_LinhaEcu.Tempo_Takt);
       "DB211_DadosScada".Ecu.StopTime := DINT_TO_INT(#Out_LinhaEcu.Tempo_StopTime);
       "DB211_DadosScada".Ecu.Objetivo := INT_TO_BYTE(#Out_LinhaEcu.Objetivo);
       "DB211_DadosScada".Ecu.Atual := INT_TO_BYTE(#Out_LinhaEcu.Atual);
       "DB211_DadosScada".Ecu.TempoRetornoParada := DINT_TO_INT(#Out_LinhaEcu.TempoRetornoParada);
       //"DB600_DadosScada".Ecu.Andon := #In_DadosEcu.ANDON;
       //"DB600_DadosScada".Ecu.Emergencia := #In_DadosEcu.EMERGENCY;
       "DB211_DadosScada".Ecu.CorDeTela := #Out_LinhaEcu.CorDeTela;
       "DB211_DadosScada".Ecu.NumMensagem := INT_TO_BYTE(#Out_LinhaEcu.NumMensagem);






   END_REGION

   //Realiza o filtro dos dados dos AGVs
   REGION Filtragem AGVs
       #FiltroDadosAgv[0](In:=#In_DadosEcu.Dados_Agv[0],
                         Out_Sinais=>"DB211_DadosScada".AGV[0].Sinais,
                         Out_Posto=>"DB211_DadosScada".AGV[0].Posto,
                         Out_Comando=>"DB211_DadosScada".AGV[0].Comando,
                         Out_Velocidade=>"DB211_DadosScada".AGV[0].Velocidade,
                         Out_Processo=>"DB211_DadosScada".AGV[0].Processo,
                         Out_VelAtual=>"DB211_DadosScada".AGV[0].VelAtual,
                         "Out_Erros.Agv"=>"DB211_DadosScada".AGV[0]."Erros.Agv",
                         "Out_Erros.Pgv"=>"DB211_DadosScada".AGV[0]."Erros.Pgv",
                         "Out_Erros.MotorPasso"=>"DB211_DadosScada".AGV[0]."Erros.MotorPasso");

      #FiltroDadosAgv[1](In := #In_DadosEcu.Dados_Agv[1],
                         Out_Sinais => "DB211_DadosScada".AGV[1].Sinais,
                         Out_Posto => "DB211_DadosScada".AGV[1].Posto,
                         Out_Comando => "DB211_DadosScada".AGV[1].Comando,
                         Out_Velocidade => "DB211_DadosScada".AGV[1].Velocidade,
                         Out_Processo => "DB211_DadosScada".AGV[1].Processo,
                         Out_VelAtual => "DB211_DadosScada".AGV[1].VelAtual,
                         "Out_Erros.Agv" => "DB211_DadosScada".AGV[1]."Erros.Agv",
                         "Out_Erros.Pgv" => "DB211_DadosScada".AGV[1]."Erros.Pgv",
                         "Out_Erros.MotorPasso" => "DB211_DadosScada".AGV[1]."Erros.MotorPasso");

      #FiltroDadosAgv[2](In := #In_DadosEcu.Dados_Agv[2],
                         Out_Sinais => "DB211_DadosScada".AGV[2].Sinais,
                         Out_Posto => "DB211_DadosScada".AGV[2].Posto,
                         Out_Comando => "DB211_DadosScada".AGV[2].Comando,
                         Out_Velocidade => "DB211_DadosScada".AGV[2].Velocidade,
                         Out_Processo => "DB211_DadosScada".AGV[2].Processo,
                         Out_VelAtual => "DB211_DadosScada".AGV[2].VelAtual,
                         "Out_Erros.Agv" => "DB211_DadosScada".AGV[2]."Erros.Agv",
                         "Out_Erros.Pgv" => "DB211_DadosScada".AGV[2]."Erros.Pgv",
                         "Out_Erros.MotorPasso" => "DB211_DadosScada".AGV[2]."Erros.MotorPasso");

      #FiltroDadosAgv[3](In := #In_DadosEcu.Dados_Agv[3],
                         Out_Sinais => "DB211_DadosScada".AGV[3].Sinais,
                         Out_Posto => "DB211_DadosScada".AGV[3].Posto,
                         Out_Comando => "DB211_DadosScada".AGV[3].Comando,
                         Out_Velocidade => "DB211_DadosScada".AGV[3].Velocidade,
                         Out_Processo => "DB211_DadosScada".AGV[3].Processo,
                         Out_VelAtual => "DB211_DadosScada".AGV[3].VelAtual,
                         "Out_Erros.Agv" => "DB211_DadosScada".AGV[3]."Erros.Agv",
                         "Out_Erros.Pgv" => "DB211_DadosScada".AGV[3]."Erros.Pgv",
                         "Out_Erros.MotorPasso" => "DB211_DadosScada".AGV[3]."Erros.MotorPasso");

      #FiltroDadosAgv[4](In := #In_DadosEcu.Dados_Agv[4],
                         Out_Sinais => "DB211_DadosScada".AGV[4].Sinais,
                         Out_Posto => "DB211_DadosScada".AGV[4].Posto,
                         Out_Comando => "DB211_DadosScada".AGV[4].Comando,
                         Out_Velocidade => "DB211_DadosScada".AGV[4].Velocidade,
                         Out_Processo => "DB211_DadosScada".AGV[4].Processo,
                         Out_VelAtual => "DB211_DadosScada".AGV[4].VelAtual,
                         "Out_Erros.Agv" => "DB211_DadosScada".AGV[4]."Erros.Agv",
                         "Out_Erros.Pgv" => "DB211_DadosScada".AGV[4]."Erros.Pgv",
                         "Out_Erros.MotorPasso" => "DB211_DadosScada".AGV[4]."Erros.MotorPasso");

      #FiltroDadosAgv[5](In := #In_DadosEcu.Dados_Agv[5],
                         Out_Sinais => "DB211_DadosScada".AGV[5].Sinais,
                         Out_Posto => "DB211_DadosScada".AGV[5].Posto,
                         Out_Comando => "DB211_DadosScada".AGV[5].Comando,
                         Out_Velocidade => "DB211_DadosScada".AGV[5].Velocidade,
                         Out_Processo => "DB211_DadosScada".AGV[5].Processo,
                         Out_VelAtual => "DB211_DadosScada".AGV[5].VelAtual,
                         "Out_Erros.Agv" => "DB211_DadosScada".AGV[5]."Erros.Agv",
                         "Out_Erros.Pgv" => "DB211_DadosScada".AGV[5]."Erros.Pgv",
                         "Out_Erros.MotorPasso" => "DB211_DadosScada".AGV[5]."Erros.MotorPasso");
      #FiltroDadosAgv[6](In := #In_DadosEcu.Dados_Agv[6],
                         Out_Sinais => "DB211_DadosScada".AGV[6].Sinais,
                         Out_Posto => "DB211_DadosScada".AGV[6].Posto,
                         Out_Comando => "DB211_DadosScada".AGV[6].Comando,
                         Out_Velocidade => "DB211_DadosScada".AGV[6].Velocidade,
                         Out_Processo => "DB211_DadosScada".AGV[6].Processo,
                         Out_VelAtual => "DB211_DadosScada".AGV[6].VelAtual,
                         "Out_Erros.Agv" => "DB211_DadosScada".AGV[6]."Erros.Agv",
                         "Out_Erros.Pgv" => "DB211_DadosScada".AGV[6]."Erros.Pgv",
                         "Out_Erros.MotorPasso" => "DB211_DadosScada".AGV[6]."Erros.MotorPasso");
      #FiltroDadosAgv[7](In := #In_DadosEcu.Dados_Agv[7],
                         Out_Sinais => "DB211_DadosScada".AGV[7].Sinais,
                         Out_Posto => "DB211_DadosScada".AGV[7].Posto,
                         Out_Comando => "DB211_DadosScada".AGV[7].Comando,
                         Out_Velocidade => "DB211_DadosScada".AGV[7].Velocidade,
                         Out_Processo => "DB211_DadosScada".AGV[7].Processo,
                         Out_VelAtual => "DB211_DadosScada".AGV[7].VelAtual,
                         "Out_Erros.Agv" => "DB211_DadosScada".AGV[7]."Erros.Agv",
                         "Out_Erros.Pgv" => "DB211_DadosScada".AGV[7]."Erros.Pgv",
                         "Out_Erros.MotorPasso" => "DB211_DadosScada".AGV[7]."Erros.MotorPasso");
      #FiltroDadosAgv[8](In := #In_DadosEcu.Dados_Agv[8],
                         Out_Sinais => "DB211_DadosScada".AGV[8].Sinais,
                         Out_Posto => "DB211_DadosScada".AGV[8].Posto,
                         Out_Comando => "DB211_DadosScada".AGV[8].Comando,
                         Out_Velocidade => "DB211_DadosScada".AGV[8].Velocidade,
                         Out_Processo => "DB211_DadosScada".AGV[8].Processo,
                         Out_VelAtual => "DB211_DadosScada".AGV[8].VelAtual,
                         "Out_Erros.Agv" => "DB211_DadosScada".AGV[8]."Erros.Agv",
                         "Out_Erros.Pgv" => "DB211_DadosScada".AGV[8]."Erros.Pgv",
                         "Out_Erros.MotorPasso" => "DB211_DadosScada".AGV[8]."Erros.MotorPasso");

      #FiltroDadosAgv[9](In := #In_DadosEcu.Dados_Agv[9],
                         Out_Sinais => "DB211_DadosScada".AGV[9].Sinais,
                         Out_Posto => "DB211_DadosScada".AGV[9].Posto,
                         Out_Comando => "DB211_DadosScada".AGV[9].Comando,
                         Out_Velocidade => "DB211_DadosScada".AGV[9].Velocidade,
                         Out_Processo => "DB211_DadosScada".AGV[9].Processo,
                         Out_VelAtual => "DB211_DadosScada".AGV[9].VelAtual,
                         "Out_Erros.Agv" => "DB211_DadosScada".AGV[9]."Erros.Agv",
                         "Out_Erros.Pgv" => "DB211_DadosScada".AGV[9]."Erros.Pgv",
                         "Out_Erros.MotorPasso" => "DB211_DadosScada".AGV[9]."Erros.MotorPasso");
   END_REGION
END_FUNCTION_BLOCK

FUNCTION_BLOCK "FB202_FiltroDados_TaktAgvs"   // FB202, SCL
TITLE = FB202_FiltroDados_TaktAgvs
{ S7_Optimized_Access := 'TRUE' }
VERSION : 0.1
// FB202_FiltroDados_TaktAgvs
   VAR_INPUT
      In_DadosEcu : "Central.Database";
      In_Turno : Struct
         Turnos : Array[0..2] of Struct
            Inicio : Date_And_Time;
            Fim : Date_And_Time;
            Objetivo : Int;
            DiasDaSemana : Array[0..6] of Bool;
            Paradas : Array[0..5] of Struct
               Inicio : Date_And_Time;
               Fim : Date_And_Time;
            END_STRUCT;
            HE_Inicio : Date_And_Time;
            HE_Fim : Date_And_Time;
         END_STRUCT;
      END_STRUCT;
   END_VAR
   VAR_OUTPUT
      Out_LinhaEcu : Struct
         Tempo_Takt : DInt;
         Tempo_StopTime : DInt;
         Objetivo : Int;
         Atual : Int;
         LinhaParada : Bool;
         TempoRetornoParada : DInt;
         LinhaRodando : Bool;
         Andons : Array[0..8] of Bool;
         CorDeTela : Byte;
         DirectRun : Real;
         SaldoDoTurno : Int;
         AndonOn : Int;
         Paradas : Array[0..1] of Struct
            Inicio : Time_Of_Day;
            Fim : Time_Of_Day;
            Posto : Int;
            ValorTimer : Int;
            ValorTimerFim : Int;
         END_STRUCT;
         NumMensagem : Int;
         Emergencias : Array[0..8] of Bool;
      END_STRUCT;
      Out_MensagemEcu : String;
   END_VAR
   VAR
      S_DateTime : Date_And_Time;
      S_CounterFor : Int;
      S_CounterFor_1 : Int;
      S_Turnos : Array[0..2] of Struct
         Paradas : Array[0..6] of Bool;
         ContagemRetorno : Array[0..6] of DInt;
      END_STRUCT;
      S_ForaDeTurno : Bool;
      S_TempoRetorno : Int;
      S_Hora : Time_Of_Day;
   END_VAR
   VAR_TEMP
      Err : Int;
   END_VAR
BEGIN

   (*
       ESTE BLOCO REALIZA O FILTRO DAS INFORMAÇÕES DO TAKT, EXEMPLOS: TROCA DA COR DA TELA, MENSAGENS NA TELA E ETC
   *)


   // Converte o sinal de andon de byte para boolean
   REGION Valores ANDON
       // Converte o sinal de andon de byte para boolean
       #Out_LinhaEcu.Andons[0] := #In_DadosEcu.Dados_Takt.Andons[0];
       #Out_LinhaEcu.Andons[1] := #In_DadosEcu.Dados_Takt.Andons[1];
       #Out_LinhaEcu.Andons[2] := #In_DadosEcu.Dados_Takt.Andons[2];
       #Out_LinhaEcu.Andons[3] := #In_DadosEcu.Dados_Takt.Andons[3];
       #Out_LinhaEcu.Andons[4] := #In_DadosEcu.Dados_Takt.Andons[4];
       #Out_LinhaEcu.Andons[5] := #In_DadosEcu.Dados_Takt.Andons[5];
       #Out_LinhaEcu.Andons[6] := #In_DadosEcu.Dados_Takt.Andons[6];
       #Out_LinhaEcu.Andons[7] := #In_DadosEcu.Dados_Takt.Andons[7];
   END_REGION

   // Converte o sinal de emergencia de byte para boolean
   REGION Valores Emergencia
       // Converte o sinal de emergencia de byte para boolean
       #Out_LinhaEcu.Emergencias[0] := #In_DadosEcu.Dados_Agv[0].Emergencia;
       #Out_LinhaEcu.Emergencias[1] := #In_DadosEcu.Dados_Agv[1].Emergencia;
       #Out_LinhaEcu.Emergencias[2] := #In_DadosEcu.Dados_Agv[2].Emergencia;
       #Out_LinhaEcu.Emergencias[3] := #In_DadosEcu.Dados_Agv[3].Emergencia;
       #Out_LinhaEcu.Emergencias[4] := #In_DadosEcu.Dados_Agv[4].Emergencia;
       #Out_LinhaEcu.Emergencias[5] := #In_DadosEcu.Dados_Agv[5].Emergencia;
       #Out_LinhaEcu.Emergencias[6] := #In_DadosEcu.Dados_Agv[6].Emergencia;
       #Out_LinhaEcu.Emergencias[7] := #In_DadosEcu.Dados_Agv[7].Emergencia;
   END_REGION

   //Realiza a leitura da hora atual do CLP
   REGION HoraAtual

       //Realiza a leitura da hora atual do CLP

       #Err := RD_LOC_T(#S_DateTime);

   END_REGION

   //Verifica se a linha esta em turno, caso não esteja retorno o tempo necessario para a linha voltar a rodar
   REGION LinhaEmTurno
       FOR #S_CounterFor := 0 TO 2 DO
           //Verifica se está em turno
           IF #In_Turno.Turnos[#S_CounterFor].Inicio >= #S_DateTime AND #S_DateTime <= #In_Turno.Turnos[#S_CounterFor].Fim THEN
               //Verifica se existe alguma parada programada
               FOR #S_CounterFor_1 := 0 TO 5 DO
                   IF #In_Turno.Turnos[#S_CounterFor].Paradas[#S_CounterFor_1].Inicio >= #S_DateTime
                       AND #S_DateTime <= #In_Turno.Turnos[#S_CounterFor].Paradas[#S_CounterFor_1].Fim THEN

                       #S_Turnos[#S_CounterFor].Paradas[#S_CounterFor_1] := 1;
                       #S_Turnos[#S_CounterFor].ContagemRetorno[#S_CounterFor_1] := TOD_TO_DINT(DT_TO_TOD(#S_DateTime - (#In_Turno.Turnos[#S_CounterFor].Paradas[#S_CounterFor_1].Fim - #In_Turno.Turnos[#S_CounterFor].Paradas[#S_CounterFor_1].Inicio)));
                   ELSE
                       #S_Turnos[#S_CounterFor].ContagemRetorno[#S_CounterFor_1] := 0;
                       #S_Turnos[#S_CounterFor].Paradas[#S_CounterFor_1] := 0;

                   END_IF;

                   #S_Turnos[#S_CounterFor].Paradas[6] := 0; // Em turno
                   #S_Turnos[#S_CounterFor].ContagemRetorno[6] := 0;
               END_FOR;
           ELSE
               #S_Turnos[#S_CounterFor].Paradas[6] := 1; // Fora de turno
               #S_Turnos[#S_CounterFor].ContagemRetorno[6] := #S_DateTime - #In_Turno.Turnos[#S_CounterFor].Paradas[#S_CounterFor_1].Inicio; // Quantidade de tempo restante para reiniciar o novo turno
           END_IF;

       END_FOR;

       #S_ForaDeTurno := #S_Turnos[0 AND 1 AND 2].Paradas[0 AND 1 AND 2 AND 3 AND 4 AND 5 AND 6];
       #S_TempoRetorno := #S_Turnos[0 AND 1 AND 2].ContagemRetorno[0 AND 1 AND 2 AND 3 AND 4 AND 5 AND 6];
   END_REGION

   REGION VerificaEmTurno
       #S_Hora := DT_TO_TOD(#S_DateTime);
       IF #S_Hora > TOD#17:00:00  THEN
           #S_TempoRetorno := (TOD_TO_INT(TOD#07:00:00)/100 - TOD_TO_INT(#S_Hora)/100);
           #S_ForaDeTurno := 1;
       ELSE
           #S_TempoRetorno := 0;
           #S_ForaDeTurno := 0;
       END_IF;


   END_REGION




   // Realiza a analise de todos os dados e troca a cor da tela
   REGION DefiniçãoCorDaTela
       // 1 - Tela Amarela (Necessario ajuda em algum posto e não estourou o tempo do TAKT)
       IF ((#Out_LinhaEcu.Andons[0] OR #Out_LinhaEcu.Andons[1] OR #Out_LinhaEcu.Andons[3] OR #Out_LinhaEcu.Andons[4] OR
           #Out_LinhaEcu.Andons[5] OR #Out_LinhaEcu.Andons[6] OR #Out_LinhaEcu.Andons[7]) AND (#In_DadosEcu.Dados_Takt.Tempo_Takt > 0)) AND NOT #S_ForaDeTurno THEN
           #Out_LinhaEcu.CorDeTela := 1;

           // 2 - Tela Vermelho (Necessario ajuda em algum posto e estourou o tempo do TAKT)
       ELSIF (((#Out_LinhaEcu.Andons[0] OR #Out_LinhaEcu.Andons[1] OR #Out_LinhaEcu.Andons[3] OR #Out_LinhaEcu.Andons[4] OR
           #Out_LinhaEcu.Andons[5] OR #Out_LinhaEcu.Andons[6] OR #Out_LinhaEcu.Andons[7]) AND (#In_DadosEcu.Dados_Takt.Tempo_Takt <= 0)) OR
           (#Out_LinhaEcu.Emergencias[0] OR #Out_LinhaEcu.Emergencias[1] OR #Out_LinhaEcu.Emergencias[3] OR  #Out_LinhaEcu.Emergencias[4] OR
           (*#Out_LinhaEcu.Emergencias[5] OR *) #Out_LinhaEcu.Emergencias[6] OR #Out_LinhaEcu.Emergencias[7])) AND NOT #S_ForaDeTurno THEN
           #Out_LinhaEcu.CorDeTela := 2;

           //3 - Tela Azul - (Aguardando inicio de turno/Volta da refeição)
       ELSIF #S_ForaDeTurno THEN
           #Out_LinhaEcu.CorDeTela := 3;

           //4 - Tela Laranja - (Aguardando retirada do produto)
       ELSIF (#Out_LinhaEcu.Andons[7]) AND NOT #S_ForaDeTurno THEN
           #Out_LinhaEcu.CorDeTela:= 4;
           //0 - Tela Branca/Preta (Tudo Ok)
       ELSE
           #Out_LinhaEcu.CorDeTela := 0;
       END_IF;


   END_REGION

   // Realiza a analise de todos os dados e escreve a mensagem na tela 
   REGION Mensagens

       IF (#Out_LinhaEcu.Emergencias[0] OR #Out_LinhaEcu.Emergencias[1] OR #Out_LinhaEcu.Emergencias[2] OR #Out_LinhaEcu.Emergencias[3] OR  #Out_LinhaEcu.Emergencias[4] OR
           (*#Out_LinhaEcu.Emergencias[5] OR *) #Out_LinhaEcu.Emergencias[6] OR #Out_LinhaEcu.Emergencias[7]) AND NOT #S_ForaDeTurno THEN

           // Sinal de EMERGÊNCIA  do posto 1
           IF #Out_LinhaEcu.Emergencias[0] THEN
               #Out_LinhaEcu.NumMensagem := 1;
               #Out_MensagemEcu := CONCAT(IN1 := 'EMERGÊNCIA DO AGV 1 ACIONADO NO POSTO ', IN2 := INT_TO_STRING(#In_DadosEcu.Dados_Agv[0].Posto));
               // Sinal de EMERGÊNCIA  do posto 2
           ELSIF #Out_LinhaEcu.Emergencias[1] THEN
               #Out_LinhaEcu.NumMensagem := 2;
               #Out_MensagemEcu := CONCAT(IN1 := 'EMERGÊNCIA DO AGV 2 ACIONADO NO POSTO ', IN2 := INT_TO_STRING(#In_DadosEcu.Dados_Agv[0].Posto));

               // Sinal de EMERGÊNCIA  do posto 3
           ELSIF #Out_LinhaEcu.Emergencias[2] THEN
               #Out_LinhaEcu.NumMensagem := 3;
               #Out_MensagemEcu := CONCAT(IN1 := 'EMERGÊNCIA DO AGV 3 ACIONADO NO POSTO ', IN2 := INT_TO_STRING(#In_DadosEcu.Dados_Agv[0].Posto));

               // Sinal de EMERGÊNCIA  do posto 4
           ELSIF #Out_LinhaEcu.Emergencias[3] THEN
               #Out_LinhaEcu.NumMensagem := 4;
               #Out_MensagemEcu := CONCAT(IN1 := 'EMERGÊNCIA DO AGV 4 ACIONADO NO POSTO ', IN2 := INT_TO_STRING(#In_DadosEcu.Dados_Agv[0].Posto));

               // Sinal de EMERGÊNCIA  do posto 5
           ELSIF #Out_LinhaEcu.Emergencias[4] AND "AlwaysFALSE" THEN
               #Out_LinhaEcu.NumMensagem := 5;
               #Out_MensagemEcu := CONCAT(IN1 := 'EMERGÊNCIA DO AGV 5 ACIONADO NO POSTO ', IN2 := INT_TO_STRING(#In_DadosEcu.Dados_Agv[0].Posto));

               // Sinal de EMERGÊNCIA  do posto 6
           ELSIF #Out_LinhaEcu.Emergencias[5] AND "AlwaysFALSE" THEN
               #Out_LinhaEcu.NumMensagem := 6;
               #Out_MensagemEcu := CONCAT(IN1 := 'EMERGÊNCIA DO AGV 6 ACIONADO NO POSTO ', IN2 := INT_TO_STRING(#In_DadosEcu.Dados_Agv[0].Posto));

               // Sinal de EMERGÊNCIA  do posto 7
           ELSIF #Out_LinhaEcu.Emergencias[6] THEN
               #Out_LinhaEcu.NumMensagem := 7;
               #Out_MensagemEcu := CONCAT(IN1 := 'EMERGÊNCIA DO AGV 7 ACIONADO NO POSTO ', IN2 := INT_TO_STRING(#In_DadosEcu.Dados_Agv[0].Posto));

               // Sinal de EMERGÊNCIA  do posto 8
           ELSIF #Out_LinhaEcu.Emergencias[7] THEN
               #Out_LinhaEcu.NumMensagem := 8;
               #Out_MensagemEcu := CONCAT(IN1 := 'EMERGÊNCIA DO AGV 8 ACIONADO NO POSTO ', IN2 := INT_TO_STRING(#In_DadosEcu.Dados_Agv[0].Posto));

           END_IF;

       ELSIF (#Out_LinhaEcu.Andons[0] OR #Out_LinhaEcu.Andons[1] OR #Out_LinhaEcu.Andons[2]OR #Out_LinhaEcu.Andons[3] OR #Out_LinhaEcu.Andons[4] OR
           #Out_LinhaEcu.Andons[5] OR #Out_LinhaEcu.Andons[6] OR #Out_LinhaEcu.Andons[7]) AND NOT #S_ForaDeTurno THEN

           // Sinal de andon do posto 1
           IF #Out_LinhaEcu.Andons[0] THEN
               #Out_LinhaEcu.NumMensagem := 9;
               #Out_MensagemEcu := 'AGUARDANDO ENTRADA DO PRODUTO NO POSTO 1';

               // Sinal de andon do posto 2
           ELSIF #Out_LinhaEcu.Andons[1] THEN
               #Out_LinhaEcu.NumMensagem := 10;
               #Out_MensagemEcu := 'NECESSARIO AJUDA NO POSTO 2';

               // Sinal de andon do posto 3
           ELSIF #Out_LinhaEcu.Andons[2] THEN
               #Out_LinhaEcu.NumMensagem := 11;
               #Out_MensagemEcu := 'NECESSARIO AJUDA NO POSTO 3';

               // Sinal de andon do posto 4
           ELSIF #Out_LinhaEcu.Andons[3] THEN
               #Out_LinhaEcu.NumMensagem := 12;
               #Out_MensagemEcu := 'NECESSARIO AJUDA NO POSTO 4';

               // Sinal de andon do posto 5
           ELSIF #Out_LinhaEcu.Andons[4] THEN
               #Out_LinhaEcu.NumMensagem := 13;
               #Out_MensagemEcu := 'NECESSARIO AJUDA NO POSTO 5';

